Yaskawa INFORM job: SKRZYNIA_5140_0_STOPNI_2OBR_NEW.JBI

/JOB
//NAME SKRZYNIA_5140_0_STOPNI_2OBR_NEW
///FOLDERNAME 02-SKRZYNIE_JOBS
//POS
///NPOS 730,730,0,52,0,0
///TOOL 0
///POSTYPE PULSE
///PULSE
C00000=1055,-24125,84372,288,19725,204
C00001=0,-15438,65714,0,-68532,0
C00002=4718,-16587,59952,3396,-65485,-935
C00003=32997,-21499,42555,27623,-61436,21376
C00004=31759,-20688,42932,26837,-60850,21559
C00005=28987,-21156,42712,24818,-60442,22222
C00006=33447,-21964,42352,27886,-61721,21330
C00007=37687,-23357,41794,30651,-63289,20620
C00008=38979,-19018,48057,32961,-64962,20678
C00009=37261,-18075,48526,31902,-64209,20901
C00010=35830,-17198,48994,31015,-63571,21092
C00011=34080,-17614,48768,29780,-63290,21485
C00012=37261,-18075,48526,31902,-64209,20901
C00013=47373,-21912,40596,41149,-66086,26950
C00014=4718,-16587,59952,3396,-65485,-935
C00015=32997,-21499,42555,27623,-61436,21376
C00016=31759,-20688,42932,26837,-60850,21559
C00017=28987,-21156,42712,24818,-60442,22222
C00018=33447,-21964,42352,27886,-61721,21330
C00019=37687,-23357,41794,30651,-63289,20620
C00020=38979,-19018,48057,32961,-64962,20678
C00021=37261,-18075,48526,31902,-64209,20901
C00022=35830,-17198,48994,31015,-63571,21092
C00023=34080,-17614,48768,29780,-63290,21485
C00024=37261,-18075,48526,31902,-64209,20901
C00025=47373,-21912,40596,41149,-66086,26950
C00026=45033,-20851,41104,39798,-65001,27223
C00027=42790,-19693,41704,38494,-63946,27495
C00028=41070,-20182,41442,37324,-63566,27891
C00029=45033,-20851,41104,39798,-65001,27223
C00030=45033,-20851,41104,39798,-65001,27223
C00031=59624,-29540,14278,64846,-60867,16042
C00032=57357,-28542,14780,63940,-59509,16120
C00033=56188,-29140,14476,63237,-58995,16387
C00034=59588,-29370,14363,64862,-60819,16012
C00035=62924,-29779,15793,65870,-63073,16252
C00036=59724,-28781,16276,64511,-61238,16415
C00037=57764,-27936,16704,63709,-60078,16488
C00038=56408,-28589,16373,62897,-59486,16787
C00039=59724,-28781,16276,64511,-61238,16415
C00040=87562,-48087,-13810,78020,-75252,11220
C00041=10104,-46603,4759,11228,-37390,-5046
C00042=0,-52280,40443,0,6876,0
C00043=1529,-42140,58025,-5964,2417,3265
C00044=0,-38374,23626,-1605,-51738,268
C00045=45044,-23015,37260,35797,-71879,25522
C00046=39973,-29571,18873,35060,-63052,24165
C00047=38620,-28701,19269,34339,-62304,24363
C00048=36409,-29254,19014,32896,-61805,24958
C00049=44451,-29039,21934,37281,-65892,23702
C00050=49472,-39353,6917,53118,-50908,20251
C00051=45058,-39356,3832,51653,-47640,20099
C00052=42883,-38319,4163,50577,-46309,20295
C00053=40255,-38926,3967,48502,-45334,21060
C00054=46774,-39679,3737,52663,-48537,19827
C00055=48708,-40455,3517,53615,-49689,19657
C00056=43798,-39237,3871,50850,-47027,20335
C00057=41951,-38324,4161,49930,-45891,20507
C00058=39836,-38844,3994,48234,-45126,21137
C00059=48489,-40338,3551,53521,-49551,19665
C00060=48489,-40338,3551,53521,-49551,19665
C00061=44432,-39026,3936,51363,-47247,20139
C00062=42487,-38069,4248,50403,-46050,20315
C00063=39061,-38795,4009,47695,-44769,21310
C00064=44432,-39026,3936,51363,-47247,20139
C00065=45358,-49480,-3557,50155,-49322,21260
C00066=1817,-44984,2816,-3462,-45659,1296
C00067=1445,-28771,30219,-502,-63201,-220
C00068=1148,-56354,34370,-22,3827,-10
C00069=0,-52280,40443,0,6876,0
C00070=0,-49898,44897,0,-65513,0
C00071=52002,-27630,35066,40617,-70496,28619
C00072=38179,-24916,32897,32855,-63545,30206
C00073=36484,-23889,33369,31863,-62698,30449
C00074=33804,-24434,33113,30025,-62179,31112
C00075=38179,-24916,32897,32855,-63545,30206
C00076=78369,-41260,16071,67181,-65880,21417
C00077=137,-45861,52341,97,-67596,-14
C00078=-31499,-58302,-23356,15027,12889,-13082
C00079=-52768,-43016,-26078,18373,38595,-18774
C00080=-89470,-32103,-32973,29905,69139,-31512
C00081=-68838,-26884,-24872,16972,64732,-23076
C00082=-53036,-11528,-12218,12363,64665,-17409
C00083=-51536,-9474,-10276,11905,64649,-16876
C00084=-51739,-9114,-7787,12104,63269,-17104
C00085=-53036,-11528,-12218,12363,64665,-17409
C00086=-17541,-26226,-24397,927,59032,-5038
C00087=-17541,-26226,-24397,927,59032,-5038
C00088=-16950,-23991,-22741,715,59568,-4818
C00089=-17036,-23563,-20101,755,58071,-4857
C00090=-17541,-26226,-24397,927,59032,-5038
C00091=34102,-23192,-21614,-15638,64271,13209
C00092=33423,-21885,-20599,-15423,64418,12942
C00093=32426,-19856,-18975,-15106,64629,12551
C00094=32578,-19611,-17013,-15290,63535,12762
C00095=33423,-21885,-20599,-15423,64418,12942
C00096=59339,-6070,-6417,-20979,72191,20891
C00097=59339,-6070,-6417,-20979,72191,20891
C00098=57897,-4256,-4562,-20702,71913,20431
C00099=58108,-3992,-2506,-20878,70835,20713
C00100=59339,-6070,-6417,-20979,72191,20891
C00101=42744,-35904,-30225,-18322,62562,16651
C00102=-53036,-11528,-12218,12363,64665,-17409
C00103=-77982,-26538,-29134,27151,66629,-27745
C00104=-70983,-8594,-1966,26503,59809,-49670
C00105=-80152,19776,40785,37351,72704,-50428
C00106=-79984,20154,42529,37516,71911,-50638
C00107=-79233,18397,40079,37458,71885,-50340
C00108=-79984,20154,42529,37516,71911,-50638
C00109=-73519,23289,38838,28890,77081,-45618
C00110=-73519,24511,42682,29072,75582,-46027
C00111=-73519,23289,38838,28890,77081,-45618
C00112=-88897,15706,42282,50101,71325,-56974
C00113=-88897,15706,42282,50101,71325,-56974
C00114=-87612,12343,37838,50071,70996,-56519
C00115=-85283,14202,40272,50301,69633,-56165
C00116=-87338,12550,38107,50098,70839,-56476
C00117=-84952,-1789,13569,34660,47724,-58955
C00118=-67641,-1674,11109,10330,44856,-44725
C00119=-66443,961,13975,9688,44721,-44210
C00120=-67641,-1674,11109,10330,44856,-44725
C00121=-67641,-376,15347,10694,42950,-44967
C00122=-67641,-1674,11109,10330,44856,-44725
C00123=-79040,417,20398,15965,28992,-57786
C00124=-76655,5212,30978,15501,25024,-57306
C00125=-76655,6949,35816,16758,23084,-57955
C00126=-76655,5212,30978,15501,25024,-57306
C00127=-74761,6919,33010,13466,24593,-56049
C00128=-80460,-2874,12270,15804,32253,-57809
C00129=-61258,-29124,-13156,26560,43617,-22150
C00130=-30420,-40507,-29240,27153,53235,15188
C00131=-18589,-38725,-21450,23338,47896,18931
C00132=-17722,-35233,-16455,23322,46926,19051
C00133=-17722,-33749,-12435,23948,45421,18620
C00134=-17722,-33892,-12819,23887,45564,18661
C00135=-16677,-31133,-11209,23138,46167,19311
C00136=-17819,-35820,-17540,23246,47228,19090
C00137=-74104,-11494,-6266,31916,75042,4269
C00138=-71226,-7329,2631,32115,71468,4273
C00139=-71226,-6504,5446,32343,70365,3922
C00140=-71226,-6611,5086,32313,70505,3967
C00141=-68386,-4058,7675,32040,69573,4789
C00142=-73314,-9412,-353,32206,72648,3829
C00143=51751,-31069,-22965,-10739,49070,48663
C00144=49028,-23852,-11575,-9841,46366,47823
C00145=49028,-23004,-8935,-10039,45204,47956
C00146=49028,-23118,-9286,-10013,45357,47939
C00147=47000,-20813,-7527,-8928,45644,47024
C00148=50476,-26208,-15307,-10408,47325,48332
C00149=90602,-5375,6902,-38786,69848,59444
C00150=83174,19950,50269,-44999,67580,58220
C00151=82362,17902,47383,-44926,67511,57879
C00152=83515,19072,48341,-44798,68200,58056
C00153=78091,19382,40247,-36371,72286,52960
C00154=78091,20664,44011,-36670,70997,53443
C00155=78091,19382,40247,-36371,72286,52960
C00156=88699,7296,38566,-55615,63182,60372
C00157=86803,3068,32674,-55410,62638,59657
C00158=84852,4315,34115,-55564,61561,59330
C00159=86803,3068,32674,-55410,62638,59657
C00160=92770,-2803,21719,-53893,67577,59421
C00161=73393,-10627,10934,-27897,30744,62458
C00162=70789,-6606,18800,-27824,27830,62140
C00163=69654,-4593,20814,-26755,27596,61444
C00164=70789,-6606,18800,-27824,27830,62140
C00165=70789,-5070,23059,-29482,26284,63017
C00166=70789,-6606,18800,-27824,27830,62140
C00167=83486,-8736,6503,-27040,35338,66550
C00168=77831,-2041,26192,-25270,18452,68895
C00169=77967,1961,32070,-26860,17569,69698
C00170=77967,5243,40752,-32914,14549,72656
C00171=77967,1961,32070,-26860,17569,69698
C00172=74560,4730,35257,-21622,16551,66717
C00173=77967,1961,32070,-26860,17569,69698
C00174=81109,-22356,2664,-22493,33121,60116
C00175=86168,-49730,-13668,-23926,46819,49343
C00176=44183,-52048,-7537,-24795,46064,51426
C00177=0,-52280,40443,0,6876,0
C00178=0,-52280,40443,0,6876,0
C00179=33629,-57276,-6399,46271,-24969,-2804
C00180=75493,-63502,-64712,103874,-64610,-6298
C00181=47885,-58436,-62704,109755,-46164,-10686
C00182=43896,-60167,-65932,114356,-43302,-9311
C00183=55379,-67378,-68041,108237,-48773,-4935
C00184=62671,-64213,-64640,104431,-56093,-7372
C00185=28458,-50318,6850,47420,-25887,-3347
C00186=0,-52280,40443,0,6876,0
C00187=1055,-24125,84372,288,19725,204
C00188=0,-15438,65714,0,-68532,0
C00189=0,-15438,65714,966,-70097,42926
C00190=69988,-9219,57065,61610,-82752,27767
C00191=63113,-6157,59685,58080,-79692,28271
C00192=46673,-5697,67857,40481,-75278,29676
C00193=49770,-5379,67539,43594,-76189,29543
C00194=63113,-6157,59685,58080,-79692,28271
C00195=69988,-9219,57065,61610,-82752,27767
C00196=0,-15438,65714,966,-70097,42926
C00197=0,-15438,65714,0,-68532,0
C00198=1055,-24125,84372,288,19725,204
C00199=1055,-24125,84372,288,19725,204
C00200=0,-41971,13909,0,6774,1
C00201=-55064,-17017,13106,20113,45767,-35735
C00202=-85641,-3161,12660,31281,67420,-55579
C00203=-77611,9747,38455,32702,57795,-55547
C00204=-77611,9747,38455,32702,57795,-55547
C00205=-80481,23547,61641,37204,60115,-56891
C00206=-80479,11681,28780,33754,71138,-52780
C00207=-73572,15026,34389,33675,67405,-51294
C00208=-73572,20195,49236,35290,62248,-53161
C00209=-82806,26311,53816,38180,73291,-53604
C00210=-71695,3747,16001,30713,64750,-51022
C00211=-70421,5575,20105,30867,63066,-51036
C00212=-35543,-20105,-5144,22821,50284,-40173
C00213=-37830,-23193,-8618,23571,50957,-40982
C00214=11136,-28839,-12562,1025,41780,-20887
C00215=20486,-27077,-7346,-12554,38415,-10736
C00216=59545,-9921,5571,-27063,51925,3267
C00217=55110,-17412,-5825,-19778,50988,-2825
C00218=79390,11759,28162,-35512,71262,52960
C00219=74811,13878,33986,-35807,67493,52464
C00220=74942,18762,48004,-37392,62815,54352
C00221=76815,18630,46530,-37158,64288,54543
C00222=79390,11759,28162,-35512,71262,52960
C00223=10831,-54278,-29128,-6468,39852,-5090
C00224=-67200,-10549,24402,-3189,24913,-39001
C00225=-75122,-2194,12822,3152,39225,-43427
C00226=-77516,10189,32861,8493,33365,-45533
C00227=-75154,17575,49272,7885,27457,-44928
C00228=-68113,9932,38901,1157,28472,-40453
C00229=-67114,5383,31515,9208,32648,-43213
C00230=-66450,3998,29285,10896,33890,-43630
C00231=-66374,3101,28136,14657,35566,-44954
C00232=-66576,452,24763,27028,43375,-49112
C00233=-69928,4230,30673,35488,50431,-52676
C00234=-77050,-3138,8526,33226,61087,-51698
C00235=-67200,-10549,24402,-3189,24913,-39001
C00236=0,-52280,40443,83103,28146,-16510
C00237=99993,-20782,22705,-13349,24734,56519
C00238=67200,-10549,24402,3189,24913,39001
C00239=75122,-2194,12822,-3152,39225,43427
C00240=74323,5203,27259,-5972,33194,43789
C00241=74015,16414,48063,-6821,27325,44224
C00242=56519,1138,28747,9235,29393,33453
C00243=55467,619,28251,10155,29461,32830
C00244=56374,-724,25854,4078,30541,35419
C00245=56480,-7201,15910,-17697,38451,43334
C00246=68252,956,25699,-34035,49810,51639
C00247=77050,-3138,8526,-33226,61087,51698
C00248=67200,-10549,24402,3189,24913,39001
C00249=0,-52280,40443,-83103,28146,16510
C00250=-99993,-20782,22705,13349,24734,-56519
C00251=-91125,453,39555,30378,52425,-51131
C00252=-81425,-5449,14825,37552,56592,-47667
C00253=-81425,-10835,-2515,34915,62871,-45127
C00254=-79239,4305,16082,37593,68846,-50182
C00255=-81302,5892,27588,46359,62943,-54679
C00256=-82227,19402,59913,51524,57300,-60581
C00257=-84844,8890,27031,38640,69740,-53449
C00258=-90096,4679,14083,37467,76581,-51973
C00259=-87885,29238,52923,40761,81198,69685
C00260=-84355,23847,39024,40698,83720,72224
C00261=-81960,27335,46957,41070,80536,71891
C00262=-82643,24718,50492,48951,72637,70260
C00263=-90480,18737,31939,47254,81986,71631
C00264=-94217,10634,17426,46901,86469,-59967
C00265=-81425,-10835,-2515,34915,62871,-45127
C00266=-81425,-5449,14825,37552,56592,-47667
C00267=-94290,-610,44819,32366,49686,-53459
C00268=0,-55136,17047,60468,32096,-4233
C00269=99993,-20782,22705,-13349,24734,56519
C00270=91125,453,39555,-30378,52425,51131
C00271=81425,-5449,14825,-37552,56592,47667
C00272=81425,-10835,-2515,-34915,62871,45127
C00273=79239,4305,16082,-37593,68846,50182
C00274=83239,4964,30263,-50637,62037,57149
C00275=83991,16425,61235,-57769,55250,63273
C00276=93928,7973,40920,-53095,64494,61640
C00277=75109,22299,39152,-26915,78743,47998
C00278=79256,17348,34699,-33448,76412,88212
C00279=79932,23608,50901,-39863,71219,88955
C00280=76220,30771,63034,-41386,67395,88927
C00281=86322,16060,37848,-39554,76452,89287
C00282=87424,-1569,9538,-38190,72401,52253
C00283=81425,-10835,-2515,-34915,62871,45127
C00284=92850,-11266,9233,-39092,60986,50964
C00285=28366,-40369,19479,-5635,23506,17663
C00286=-80334,-19501,31260,21216,42469,-40219
C00287=-80621,-32280,-9061,25825,59412,-41877
C00288=-80621,-37319,-22868,24573,64555,-40576
C00289=-75108,-2453,16462,35304,60348,-42510
C00290=-72231,7240,33473,36511,55681,-43130
C00291=-35770,-19109,7486,28512,40799,-31761
C00292=-39606,-22901,-1163,28356,44724,-32188
C00293=15344,-29112,-5358,-2858,33820,-6852
C00294=13390,-24012,2637,-1527,32105,-7853
C00295=57983,-8601,15571,-27088,42703,12849
C00296=60973,-17187,4937,-27817,44388,13718
C00297=60973,-17187,4937,-27817,44388,13718
C00298=-13287,-42463,-12044,19170,31021,-23010
C00299=-17374,-21287,20534,22794,29118,-26096
C00300=13276,-20759,18622,-1911,29377,-7028
C00301=39924,-14247,19329,-14795,35999,4396
C00302=41528,-14133,18797,-15449,36702,5040
C00303=57001,-5890,26499,-21893,40771,11494
C00304=64054,-19541,3059,-29141,44956,15011
C00305=51466,-33957,-1499,-46586,51805,23434
C00306=17032,-20770,22044,-28854,30468,11088
C00307=-9868,-18638,14971,-8492,38486,-5199
C00308=-40562,-13194,19800,9508,35447,-20184
C00309=-41848,-12620,20103,10165,35810,-20773
C00310=-57278,-4046,28217,17578,39066,-27653
C00311=-71680,-19835,10874,33863,39440,-36917
C00312=-20806,-37586,-12792,9951,42782,-18031
C00313=29087,-45372,27330,-13325,19529,9021
C00314=0,-52280,40443,0,6876,0
C00315=0,-52280,40443,0,6876,0
C00316=0,-17525,61946,0,273,32004
C00317=54446,-4421,37881,-48560,57645,57448
C00318=45059,-5790,38757,-53071,45868,54447
C00319=46561,-4822,57063,-86189,40693,71736
C00320=46137,-328,57206,-69896,42561,59838
C00321=35508,-2998,35633,-40347,47515,38753
C00322=43067,2853,36106,-38598,60324,43004
C00323=45059,-5790,38757,-53071,45868,54447
C00324=54446,-4421,37881,-48560,57645,57448
C00325=0,-17525,61946,0,273,32004
C00326=0,-52280,40443,0,6876,0
C00327=0,-52280,40443,0,6876,0
C00328=0,-52280,40443,0,6876,0
C00329=0,-52280,40443,0,-42737,40640
C00330=0,-52280,40443,0,-42737,40640
C00331=64551,-35409,28076,75550,-44539,17239
C00332=49799,-25338,45366,61341,-39751,21495
C00333=45731,-22710,35392,68644,-36821,18294
C00334=37993,-24684,30723,57032,-36974,21705
C00335=37887,-25651,28733,57662,-36597,21303
C00336=43117,-27612,29118,67655,-35359,18183
C00337=39863,-22026,47404,54615,-35502,22403
C00338=0,-52277,40442,0,6872,2
C00339=0,-38538,66749,0,-898,0
C00340=0,-52280,40443,0,-79033,35417
C00341=46775,-35113,22190,42926,-67531,20697
C00342=52587,-26056,25345,47610,-66542,17970
C00343=45640,-25642,24411,43945,-63126,18913
C00344=46067,-27754,19531,44807,-62059,18176
C00345=53914,-29436,22058,48262,-67266,17843
C00346=63113,-6157,59685,58080,-79692,28271
C00347=47789,-6280,67353,41142,-75661,29541
C00348=46856,-5642,67903,40595,-75324,29647
C00349=49398,-5231,67705,43314,-76061,29572
C00350=59203,-5425,63284,53118,-78384,28542
C00351=46775,-35113,22190,42926,-67531,20697
C00352=0,-52280,40443,0,-79033,35417
C00353=0,-52280,40443,0,-61239,28081
C00354=53819,-14110,13758,-46164,60155,50576
C00355=48398,-14119,9451,-44868,59619,48162
C00356=41231,-18689,20734,-60860,39616,53092
C00357=26205,-20881,5343,-31434,40895,31963
C00358=48398,-14119,9451,-44868,59619,48162
C00359=53819,-14110,13758,-46164,60155,50576
C00360=0,-52280,40443,0,-61239,28081
C00361=404,-42897,57020,-1574,2523,869
C00362=404,-42897,57020,-1574,2523,869
C00363=0,-52280,40443,0,6876,0
C00364=-99253,-13690,44082,59847,13407,-31313
C00365=-87814,-12734,20141,45739,-14352,-64418
C00366=-86669,-6582,30812,41148,-16781,-62025
C00367=-85055,-5827,31548,44003,-17420,-63187
C00368=-85971,-6262,31124,42409,-17052,-62539
C00369=-86650,-5303,32069,41395,-16716,-62141
C00370=-94954,-14494,-1860,-7818,15857,-59130
C00371=-93142,-9291,12181,-6959,15791,-58178
C00372=-93142,-8228,15250,-7572,14488,-57881
C00373=-93142,-9291,12181,-6959,15791,-58178
C00374=-86125,-12470,22545,29004,-25567,-58412
C00375=-83883,-11340,22525,32952,-25567,-60136
C00376=-82768,-10824,22986,34487,-25904,-60776
C00377=-83883,-11340,22525,32952,-25567,-60136
C00378=-85143,-9772,23941,31487,-24966,-59556
C00379=-83883,-11340,22525,32952,-25567,-60136
C00380=-85732,-21202,11427,30682,-24763,-59235
C00381=-84150,-10929,23786,31981,-25941,-59678
C00382=-83036,-10419,24246,33504,-26268,-60308
C00383=-84150,-10929,23786,31981,-25941,-59678
C00384=-85291,-9507,25078,30650,-25411,-59154
C00385=-84150,-10929,23786,31981,-25941,-59678
C00386=-85786,-16909,14677,31743,-23900,-59790
C00387=-84150,-10498,24888,31517,-26306,-59436
C00388=-83174,-10052,25293,32841,-26587,-59984
C00389=-84150,-10498,24888,31517,-26306,-59436
C00390=-85258,-9112,26156,30226,-25800,-58928
C00391=-84150,-10498,24888,31517,-26306,-59436
C00392=-87841,-18519,13420,28367,-23534,-58339
C00393=-84845,-10773,24694,30524,-26144,-59020
C00394=-83241,-10052,25348,32714,-26598,-59924
C00395=-84150,-10465,24972,31484,-26336,-59417
C00396=-85145,-9228,26102,30329,-25881,-58963
C00397=-84150,-10465,24972,31484,-26336,-59417
C00398=-86371,-18277,13606,30568,-23951,-59265
C00399=-84931,-11946,21758,31628,-25145,-59609
C00400=-83211,-11173,22442,34044,-25650,-60618
C00401=-84345,-11688,21985,32461,-25312,-59957
C00402=-85283,-10526,23025,31366,-24861,-59525
C00403=-84345,-11688,21985,32461,-25312,-59957
C00404=-86191,-19647,12567,30467,-24278,-59187
C00405=-84870,-11108,23866,30820,-25860,-59178
C00406=-83051,-10286,24607,33321,-26381,-60213
C00407=-84345,-10877,24073,31552,-26006,-59481
C00408=-85179,-9842,25009,30582,-25619,-59100
C00409=-84345,-10877,24073,31552,-26006,-59481
C00410=-85438,-18022,14839,31140,-24818,-59429
C00411=-84247,-11820,22550,32049,-25753,-59727
C00412=-84627,-11209,23435,31382,-25751,-59435
C00413=-82990,-10465,24105,33639,-26227,-60372
C00414=-84104,-10976,23642,32111,-25899,-59738
C00415=-84898,-9998,24525,31196,-25529,-59378
C00416=-84104,-10976,23642,32111,-25899,-59738
C00417=-86610,-16845,14732,30573,-23614,-59301
C00418=-84466,-11025,23783,31488,-25891,-59466
C00419=-82824,-10273,24459,33737,-26370,-60397
C00420=-84104,-10864,23927,31990,-25993,-59674
C00421=-84789,-10021,24690,31200,-25673,-59363
C00422=-84104,-10864,23927,31990,-25993,-59674
C00423=-83806,-19585,12613,33764,-25080,-60559
C00424=-84285,-10368,25328,31127,-26432,-59250
C00425=-82780,-9675,25960,33156,-26866,-60087
C00426=-83924,-10205,25475,31619,-26533,-59453
C00427=-84478,-9530,26093,30986,-26280,-59206
C00428=-83924,-10205,25475,31619,-26533,-59453
C00429=-87149,-17993,13826,29513,-23647,-58830
C00430=-84920,-13182,20975,31162,-25481,-59361
C00431=-84012,-10708,24730,31646,-26390,-59479
C00432=-82779,-10142,25241,33309,-26748,-60166
C00433=-83711,-10572,24852,32056,-26475,-59649
C00434=-84370,-9774,25579,31305,-26170,-59356
C00435=-83711,-10572,24852,32056,-26475,-59649
C00436=-83642,-3679,42021,23358,-36761,-56118
C00437=-85886,-5975,41264,18964,-40261,-54782
C00438=-84505,-11891,22094,31989,-25448,-59736
C00439=-82884,-11162,22742,34234,-25925,-60671
C00440=-83919,-11632,22322,32811,-25616,-60079
C00441=-84723,-10654,23196,31887,-25230,-59715
C00442=-83919,-11632,22322,32811,-25616,-60079
C00443=-87348,-16035,7353,17528,-35245,-56477
C00444=-86906,-16205,7213,17977,-35365,-56684
C00445=-86616,-16813,3502,19256,-33445,-57386
C00446=-85308,-16228,3988,20718,-33648,-58082
C00447=-86244,-16649,3638,19674,-33501,-57585
C00448=-86740,-15973,4201,19194,-33277,-57362
C00449=-86244,-16649,3638,19674,-33501,-57585
C00450=-73780,-8639,20128,34258,-51705,-52097
C00451=-90965,-18271,-29411,11001,-28333,-56925
C00452=-93309,-19947,-33502,6140,-24593,-56497
C00453=-91512,-19116,-32812,8551,-24603,-57834
C00454=-92565,-19610,-33223,7138,-24591,-57051
C00455=-93003,-18716,-32476,6600,-24397,-56752
C00456=-92565,-19610,-33223,7138,-24591,-57051
C00457=-92565,-19610,-33223,7138,-24591,-57051
C00458=-95836,-54375,-51122,6031,-17685,-48210
C00459=-95836,-54375,-51122,6031,-17685,-48210
C00460=-43821,-47238,-2775,-3022,56549,-3681
C00461=-20126,-26882,59542,2406,16879,-9162
C00462=-20126,-26882,59542,2406,16879,-9162
C00463=98601,-10520,92678,4674,-40855,-9615
C00464=95537,-19831,-2695,-2933,-44471,35837
C00465=92548,-20391,-28429,-6186,-30623,55200
C00466=93192,-17848,-29686,-6005,-27810,55077
C00467=92147,-17363,-29270,-7221,-27815,55772
C00468=90371,-16495,-28521,-9286,-27856,56953
C00469=91429,-17018,-28974,-8057,-27827,56250
C00470=92033,-15799,-27911,-7415,-27588,55880
C00471=91429,-17018,-28974,-8057,-27827,56250
C00472=92548,-20391,-28429,-6186,-30623,55200
C00473=91156,-15018,-4648,-8036,-38181,54813
C00474=90585,-14766,-4428,-8565,-38201,55100
C00475=88830,-13959,-3717,-10186,-38284,55977
C00476=89897,-14456,-4157,-9202,-38230,55445
C00477=90761,-12944,-2809,-8452,-37927,55043
C00478=89897,-14456,-4157,-9202,-38230,55445
C00479=89910,-11217,67535,-9455,-58896,55399
C00480=89910,-11217,67535,-9455,-58896,55399
C00481=85786,-16735,14816,-31782,-23869,59812
C00482=84033,-13230,17727,-35008,-23968,61233
C00483=82251,-12406,18443,-37550,-24551,62308
C00484=83514,-12996,17929,-35760,-24132,61552
C00485=84258,-12095,18717,-34917,-23742,61217
C00486=83514,-12996,17929,-35760,-24132,61552
C00487=87149,-17993,13826,-29513,-23647,58830
C00488=83574,-13027,17908,-35676,-24115,61514
C00489=81915,-12248,18589,-38020,-24666,62504
C00490=83118,-12818,18089,-36330,-24263,61791
C00491=83897,-11882,18912,-35460,-23856,61445
C00492=83118,-12818,18089,-36330,-24263,61791
C00493=83806,-19585,12613,-33764,-25080,60559
C00494=83575,-13270,17698,-35618,-24145,61476
C00495=81675,-12378,18472,-38297,-24777,62607
C00496=82998,-13006,17925,-36445,-24332,61826
C00497=83876,-11958,18841,-35466,-23874,61442
C00498=82998,-13006,17925,-36445,-24332,61826
C00499=86610,-16845,14732,-30573,-23614,59301
C00500=82990,-13468,17528,-36367,-24395,61793
C00501=81406,-12724,18174,-38578,-24928,62723
C00502=82493,-13239,17725,-37070,-24559,62089
C00503=83436,-12134,18690,-36041,-24064,61684
C00504=82493,-13239,17725,-37070,-24559,62089
C00505=84814,-16043,15376,-33312,-24093,60464
C00506=83076,-13850,17202,-36172,-24411,61704
C00507=81384,-13062,17878,-38534,-24974,62698
C00508=82555,-13613,17404,-36910,-24580,62015
C00509=83566,-12434,18427,-35805,-24047,61580
C00510=82555,-13613,17404,-36910,-24580,62015
C00511=86191,-19647,12567,-30467,-24278,59187
C00512=83141,-13940,17126,-36065,-24398,61655
C00513=81467,-13161,17792,-38413,-24955,62645
C00514=82500,-13648,17375,-36975,-24607,62039
C00515=83481,-12505,18364,-35905,-24087,61617
C00516=82500,-13648,17375,-36975,-24607,62039
C00517=86371,-18277,13606,-30568,-23951,59265
C00518=83407,-14016,17058,-35697,-24309,61505
C00519=81715,-13237,17726,-38081,-24865,62509
C00520=82904,-13790,17251,-36416,-24470,61808
C00521=83686,-12878,18037,-35556,-24055,61469
C00522=82904,-13790,17251,-36416,-24470,61808
C00523=87841,-18519,13420,-28367,-23534,58339
C00524=83373,-14160,16936,-35712,-24341,61507
C00525=81692,-13388,17594,-38077,-24893,62505
C00526=82748,-13879,17174,-36603,-24542,61883
C00527=83607,-12881,18032,-35663,-24082,61515
C00528=82748,-13879,17174,-36603,-24542,61883
C00529=85786,-16909,14677,-31743,-23900,59790
C00530=83147,-14479,16665,-35944,-24472,61597
C00531=81460,-13708,17319,-38301,-25026,62591
C00532=82520,-14198,16902,-36833,-24674,61972
C00533=83571,-12989,17938,-35691,-24113,61524
C00534=82520,-14198,16902,-36833,-24674,61972
C00535=85732,-21202,11427,-30682,-24763,59235
C00536=83169,-14709,16474,-35859,-24497,61553
C00537=81172,-13798,17245,-38643,-25153,62725
C00538=82398,-14365,16763,-36952,-24745,62014
C00539=83600,-12984,17944,-35650,-24102,61504
C00540=82398,-14365,16763,-36952,-24745,62014
C00541=92346,-18713,13565,-21110,-22545,55257
C00542=83258,-14188,16907,-35850,-24389,61565
C00543=81518,-13384,17592,-38292,-24965,62594
C00544=82794,-13980,17083,-36511,-24538,61844
C00545=83714,-12912,18003,-35501,-24048,61445
C00546=82794,-13980,17083,-36511,-24538,61844
C00547=86140,-12802,12665,-93523,-10743,85795
C00548=86837,-13114,12391,-93393,-10290,85805
C00549=85030,-12289,13120,-93723,-11463,85776
C00550=86140,-12802,12665,-93523,-10743,85795
C00551=86958,-11660,13681,-94506,-10238,86349
C00552=85239,-16743,-4327,42764,21357,45785
C00553=86298,-7639,7084,25531,26453,52172
C00554=86298,-6383,11028,27162,24874,51322
C00555=86298,-7639,7084,25531,26453,52172
C00556=82295,-26986,-30576,21875,37939,54070
C00557=85045,-36869,-4353,-28502,-22832,52282
C00558=0,-24029,84339,0,19981,0
C00559=0,-24029,84339,0,19981,0
C00560=3172,-24246,80980,3465,15913,689
C00561=-86563,-26985,13879,10257,-21548,-45530
C00562=-86191,-19647,12567,30467,-24278,-59187
C00563=-83221,-13587,17636,37793,-25116,-62228
C00564=-91978,-13833,14560,12391,-18633,-51524
C00565=-94992,-13830,14285,1276,-18012,-46664
C00566=-84074,-17488,11256,38660,-23649,-62784
C00567=-73679,-33270,1000,44272,-31600,-64253
C00568=-86926,-60758,23267,6576,1160,-9545
C00569=0,-52280,40443,0,6876,0
C00570=82475,-58079,26734,835,4084,4444
C00571=97932,-26840,7691,8784,-23444,42538
C00572=87166,-16607,16322,-25365,-24201,56345
C00573=84744,-11374,21734,-29079,-24723,57922
C00574=84804,-11023,22730,-28561,-25071,57659
C00575=85100,-26994,10417,-24982,-28140,55821
C00576=0,-52280,40443,0,6876,0
C00577=0,-52280,40443,0,6876,0
C00578=-90140,-60305,18108,-2708,1721,-7625
C00579=-95594,-27428,6866,-4663,-19832,-42154
C00580=-98688,-13767,16447,-18366,-10080,-35766
C00581=-99366,-12207,13361,-76262,-4504,-7609
C00582=-98825,-14297,3352,-138105,-6872,21732
C00583=-99703,-3544,30885,-62667,-5630,-13378
C00584=-99859,-2424,20650,-157436,-17585,31647
C00585=-99057,-6525,-3028,-166156,-45024,38419
C00586=-98286,-5427,328,-166417,-43477,38616
C00587=-98488,3848,8620,-169322,-45735,38851
C00588=-99936,2884,1652,-167416,-53424,38690
C00589=-96149,-9016,-15084,-169449,-55688,40292
C00590=-90140,-60305,18108,-2708,1721,-7625
C00591=0,-52280,40443,0,6876,0
C00592=84259,-57935,27522,-3761,3673,6310
C00593=86507,-39672,4297,-27618,-16640,46340
C00594=73669,-37119,-20783,-92053,-19719,85232
C00595=86539,-20830,1725,-71850,-11773,76853
C00596=97574,-21911,-7032,-15733,6173,47170
C00597=94640,-18033,-2805,930,6039,39142
C00598=97727,-14050,2363,-13742,12741,47040
C00599=100679,-6296,-4637,-9974,40184,43946
C00600=100653,-5025,-17306,-8356,57963,47370
C00601=98357,-1060,-14638,-7161,64336,49394
C00602=99096,-3774,-7192,-7126,47828,42427
C00603=97072,-20012,-39240,-5169,57466,41015
C00604=96250,-19428,-8283,-4838,27297,37910
C00605=86507,-39672,4297,-27618,-16640,46340
C00606=84259,-57935,27522,-3761,3673,6310
C00607=0,-52280,40443,0,6876,0
C00608=0,-27933,77061,0,20812,0
C00609=0,-27933,77061,0,20812,0
C00610=0,-52280,40443,0,6876,0
C00611=-91970,-60791,14435,-3343,512,-9412
C00612=-98647,-24138,10005,-11519,-21203,-39749
C00613=-99883,-13980,22886,-11640,-25090,-40341
C00614=-99702,-9154,61728,-1148,-61809,-40243
C00615=-84328,-13042,29707,23458,-33731,-54641
C00616=-83101,-4179,39208,25894,-34785,-55667
C00617=-82881,-4330,38692,26392,-34479,-55866
C00618=-76259,-18287,26646,31659,-38322,-57579
C00619=-89741,-28009,12101,4461,-28076,-46404
C00620=-91970,-60791,14435,-3343,512,-9412
C00621=0,-52280,40443,0,6876,0
C00622=91083,-60784,14823,-9043,-825,15173
C00623=83869,-19403,12921,-33769,-24740,60260
C00624=83869,-19403,12921,-33769,-24740,60260
C00625=83932,-19538,53415,-33663,-71112,60249
C00626=83932,-19538,53415,-33663,-71112,60249
C00627=82480,-12247,21118,-35440,-26416,60009
C00628=82194,-11433,19802,-37650,-25323,61125
C00629=81904,-9374,24711,-35791,-26879,60109
C00630=79790,-20261,14917,-36681,-28829,60258
C00631=76554,-29711,-1870,-46042,-25952,65654
C00632=91083,-60784,14823,-9043,-825,15173
C00633=0,-52280,40443,0,6876,0
C00634=-91526,-60598,16699,7584,176,-13289
C00635=-81382,-25890,9219,35455,-25500,-59095
C00636=-86453,-20958,12525,30076,-22568,-57089
C00637=-86589,-16097,16237,31250,-21582,-57704
C00638=-98933,-11298,20505,-13970,-18736,-37953
C00639=-98281,-10965,21163,-11559,-18548,-39330
C00640=-85424,-18472,14402,34409,-22969,-58895
C00641=-74746,-27148,8488,44263,-29128,-62418
C00642=-81326,-27507,8265,35533,-26282,-59001
C00643=-91415,-60262,16631,7870,-73,-13734
C00644=24,-24029,84339,7,19981,5
C00645=100404,-52373,45687,-1822,14816,-5144
C00646=75939,-26469,7919,-40869,-29645,63133
C00647=81882,-22565,10470,-35355,-26404,61107
C00648=82801,-12246,21732,-34208,-26055,60642
C00649=91782,-10629,23559,-8729,-22207,49851
C00650=96500,-9524,26299,5706,-23134,43728
C00651=77262,-23244,14300,-38922,-31295,61912
C00652=78410,-22868,15324,-38001,-30064,61274
C00653=96357,-43275,13317,73005,-20942,3046
C00654=567,-24029,84339,168,19981,112
C00655=-91970,-60791,14435,-3343,512,-9412
C00656=-98991,-22833,11519,-12824,-17638,-36336
C00657=-86376,-13627,18436,38326,-18406,-58533
C00658=-85581,-10814,20279,41280,-18093,-59893
C00659=-85472,-10371,21054,41064,-18287,-59771
C00660=-86274,-24518,9978,34497,-20333,-56613
C00661=-91684,-53777,2301,20525,-9313,-33684
C00662=-67305,-55044,34987,1504,5690,-2468
C00663=0,-52280,40443,0,6876,0
C00664=77036,-56616,31288,-2531,4707,4197
C00665=84359,-28321,8817,-32860,-20485,54199
C00666=81156,-16932,14874,-39538,-26422,62851
C00667=93153,-15089,13046,-5673,-18101,48746
C00668=90780,-14174,15526,-13510,-19626,52025
C00669=77970,-27630,4721,-41834,-28549,63607
C00670=81111,-35571,7141,-33980,-21909,52006
C00671=82626,-57814,28323,-4146,3364,6346
C00672=0,-52280,40443,0,6876,0
C00673=0,-28135,76691,0,20839,0
C00674=0,-28135,76691,0,20839,0
C00675=-45332,-39712,59352,-1730,18713,2903
C00676=-94065,-8316,59352,-1730,-37754,-40387
C00677=-100331,-14895,33931,-8215,-36518,-40227
C00678=-98931,-8578,39429,-6260,-48307,-43744
C00679=-100336,-4176,46216,-7600,-55875,-44633
C00680=-93952,8947,73671,995,-68520,-43850
C00681=-98791,-3170,32594,-4861,-60761,-43748
C00682=-98640,4466,38023,-4864,-58745,-43707
C00683=-98715,-12714,-17812,-7609,-33367,-41875
C00684=-98688,-14490,-28435,-9054,-27450,-41090
C00685=-99605,-15546,-21493,-8548,-33053,-41326
C00686=-100467,-8208,-2562,-8095,-44661,-42156
C00687=-93952,8947,73671,995,-68520,-43850
C00688=-88754,54,62805,4404,-67858,-45120
C00689=-100222,-4532,45667,-7492,-55263,-44561
C00690=-100331,-14895,33931,-8215,-36518,-40227
C00691=-94065,-8316,59352,-1730,-37754,-40387
C00692=-45544,-32973,71870,-2133,15168,3033
C00693=0,-28135,76691,0,20839,0
C00694=54178,-17846,77779,596,-29686,20997
C00695=54178,-17846,77779,596,-29686,20997
C00696=99462,-18987,75418,611,-28919,20989
C00697=98707,-9390,78674,1080,-71212,38250
C00698=98768,-5182,41096,1808,-44974,38308
C00699=100431,1771,51615,3823,-56746,39115
C00700=97953,-6621,17555,2289,-50176,39420
C00701=95834,-5353,18817,760,-50052,40242
C00702=86491,-3931,18489,-13403,-48438,44853
C00703=88887,-11110,-8515,-11527,-36861,46615
C00704=88808,-13839,-20865,-13699,-30585,47852
C00705=90457,-16080,-12990,-9972,-37305,45724
C00706=97953,-6621,17555,2289,-50176,39420
C00707=100431,1771,51615,3823,-56746,39115
C00708=98768,-5182,41096,1808,-44974,38308
C00709=98707,-9390,78674,1080,-71212,38250
C00710=0,-28135,76691,0,20839,0
C00711=0,-28135,76691,0,20839,0
C00712=-91526,-60598,16699,7584,176,-13289
C00713=-81382,-25890,9219,35455,-25500,-59095
C00714=-81382,-25890,9219,35455,-25500,-59095
C00715=-85509,-13950,19358,32213,-22393,-58041
C00716=-96341,-12086,19487,-5053,-17846,-42145
C00717=-97523,-9822,24708,-8570,-19966,-40659
C00718=-84656,-25369,12054,31249,-26195,-57129
C00719=-82652,-57346,29982,2770,3944,-5064
C00720=0,-52280,40443,0,6876,0
C00721=60653,-54633,35892,-1212,5841,2035
C00722=77942,-28227,6869,-38010,-29303,61907
C00723=82500,-13648,17375,-36975,-24607,62039
C00724=80844,-11529,18736,-41531,-25394,63903
C00725=80409,-10373,22284,-40214,-26848,63104
C00726=64389,-31987,5108,-50419,-37074,66126
C00727=60653,-54633,35892,-1212,5841,2035
C00728=0,-52280,40443,0,6876,0
C00729=0,-28167,76633,0,20843,0
BC00000=413138
BC00001=413138
BC00002=295997
BC00003=264574
BC00004=264574
BC00005=264574
BC00006=264574
BC00007=233852
BC00008=284288
BC00009=284288
BC00010=284288
BC00011=284288
BC00012=284288
BC00013=356545
BC00014=388163
BC00015=356740
BC00016=356740
BC00017=356740
BC00018=356740
BC00019=356740
BC00020=407176
BC00021=407176
BC00022=407176
BC00023=407176
BC00024=407176
BC00025=479433
BC00026=479433
BC00027=479433
BC00028=479433
BC00029=479433
BC00030=530237
BC00031=530237
BC00032=530237
BC00033=530237
BC00034=530237
BC00035=601977
BC00036=601977
BC00037=601977
BC00038=601977
BC00039=601977
BC00040=601977
BC00041=522422
BC00042=522422
BC00043=671734
BC00044=689202
BC00045=689202
BC00046=689202
BC00047=689202
BC00048=689202
BC00049=689202
BC00050=726463
BC00051=726463
BC00052=726463
BC00053=726463
BC00054=726463
BC00055=782137
BC00056=782137
BC00057=782137
BC00058=782137
BC00059=782137
BC00060=850421
BC00061=850421
BC00062=850421
BC00063=850421
BC00064=850421
BC00065=850421
BC00066=823841
BC00067=797607
BC00068=755227
BC00069=755227
BC00070=915219
BC00071=914226
BC00072=914226
BC00073=914226
BC00074=914226
BC00075=914226
BC00076=914226
BC00077=922367
BC00078=927819
BC00079=927819
BC00080=927819
BC00081=943180
BC00082=943180
BC00083=943180
BC00084=943180
BC00085=943180
BC00086=943180
BC00087=943180
BC00088=943180
BC00089=943180
BC00090=943180
BC00091=943180
BC00092=943180
BC00093=943180
BC00094=943180
BC00095=943180
BC00096=943180
BC00097=943180
BC00098=943180
BC00099=943180
BC00100=943180
BC00101=943180
BC00102=943180
BC00103=943180
BC00104=943180
BC00105=943180
BC00106=943182
BC00107=943182
BC00108=943182
BC00109=943182
BC00110=943182
BC00111=943182
BC00112=943182
BC00113=943182
BC00114=943182
BC00115=943182
BC00116=943182
BC00117=943182
BC00118=943182
BC00119=943182
BC00120=943182
BC00121=943182
BC00122=943182
BC00123=943182
BC00124=943182
BC00125=943182
BC00126=943182
BC00127=943182
BC00128=943182
BC00129=943183
BC00130=943184
BC00131=943184
BC00132=943184
BC00133=943184
BC00134=943184
BC00135=943184
BC00136=943184
BC00137=943184
BC00138=943184
BC00139=943184
BC00140=943184
BC00141=943156
BC00142=943170
BC00143=943170
BC00144=943170
BC00145=943170
BC00146=943170
BC00147=943170
BC00148=943170
BC00149=943184
BC00150=943184
BC00151=943184
BC00152=943184
BC00153=943184
BC00154=943184
BC00155=943184
BC00156=943184
BC00157=943184
BC00158=943184
BC00159=943184
BC00160=943184
BC00161=943184
BC00162=943184
BC00163=943184
BC00164=943184
BC00165=943184
BC00166=943184
BC00167=943184
BC00168=943184
BC00169=943184
BC00170=943184
BC00171=943184
BC00172=943184
BC00173=943184
BC00174=911399
BC00175=884954
BC00176=838173
BC00177=838173
BC00178=727925
BC00179=734552
BC00180=750834
BC00181=750837
BC00182=811927
BC00183=811927
BC00184=760768
BC00185=744267
BC00186=744267
BC00187=413138
BC00188=413138
BC00189=413138
BC00190=408626
BC00191=408626
BC00192=408753
BC00193=347392
BC00194=408626
BC00195=408626
BC00196=413138
BC00197=413138
BC00198=413138
BC00199=505502
BC00200=893917
BC00201=915147
BC00202=918406
BC00203=918406
BC00204=918406
BC00205=918406
BC00206=935268
BC00207=935270
BC00208=935270
BC00209=935270
BC00210=935270
BC00211=935270
BC00212=935270
BC00213=935270
BC00214=935270
BC00215=935269
BC00216=935270
BC00217=935271
BC00218=935271
BC00219=935271
BC00220=935271
BC00221=935271
BC00222=935271
BC00223=930781
BC00224=906929
BC00225=936106
BC00226=936109
BC00227=936109
BC00228=936106
BC00229=936107
BC00230=936108
BC00231=936108
BC00232=936109
BC00233=936109
BC00234=936109
BC00235=906929
BC00236=835535
BC00237=835535
BC00238=906929
BC00239=936106
BC00240=936109
BC00241=936109
BC00242=936109
BC00243=936109
BC00244=936114
BC00245=936121
BC00246=936110
BC00247=936109
BC00248=906929
BC00249=835535
BC00250=835535
BC00251=872997
BC00252=918800
BC00253=938197
BC00254=938199
BC00255=938199
BC00256=938199
BC00257=938199
BC00258=938775
BC00259=938199
BC00260=952138
BC00261=952138
BC00262=952138
BC00263=952138
BC00264=952138
BC00265=938197
BC00266=918800
BC00267=872997
BC00268=873283
BC00269=835535
BC00270=872997
BC00271=918800
BC00272=938197
BC00273=938199
BC00274=938199
BC00275=938199
BC00276=938199
BC00277=938199
BC00278=938199
BC00279=938199
BC00280=938199
BC00281=938199
BC00282=938199
BC00283=938197
BC00284=918800
BC00285=849812
BC00286=864290
BC00287=883850
BC00288=922155
BC00289=922155
BC00290=922155
BC00291=922153
BC00292=922155
BC00293=922155
BC00294=922155
BC00295=922153
BC00296=922155
BC00297=914820
BC00298=922155
BC00299=922155
BC00300=922151
BC00301=922153
BC00302=922197
BC00303=922153
BC00304=922155
BC00305=922155
BC00306=922151
BC00307=922153
BC00308=922155
BC00309=922155
BC00310=922155
BC00311=922155
BC00312=918747
BC00313=805523
BC00314=697681
BC00315=697681
BC00316=697681
BC00317=733666
BC00318=758324
BC00319=767340
BC00320=794510
BC00321=816578
BC00322=794510
BC00323=758324
BC00324=733666
BC00325=697681
BC00326=697681
BC00327=697681
BC00328=841681
BC00329=841681
BC00330=884227
BC00331=901088
BC00332=895224
BC00333=896289
BC00334=924873
BC00335=936999
BC00336=921975
BC00337=887634
BC00338=824879
BC00339=507816
BC00340=507816
BC00341=552804
BC00342=552804
BC00343=551170
BC00344=493239
BC00345=491979
BC00346=285738
BC00347=285865
BC00348=285441
BC00349=256782
BC00350=258630
BC00351=552804
BC00352=507816
BC00353=507816
BC00354=507816
BC00355=531288
BC00356=531293
BC00357=591240
BC00358=531288
BC00359=507816
BC00360=507816
BC00361=507816
BC00362=507816
BC00363=848972
BC00364=861901
BC00365=963633
BC00366=963633
BC00367=963633
BC00368=963633
BC00369=963633
BC00370=963633
BC00371=963633
BC00372=963633
BC00373=963633
BC00374=963633
BC00375=963633
BC00376=963633
BC00377=963633
BC00378=963633
BC00379=963633
BC00380=902188
BC00381=895372
BC00382=895372
BC00383=895372
BC00384=895372
BC00385=895372
BC00386=840744
BC00387=840744
BC00388=840744
BC00389=840744
BC00390=840744
BC00391=840744
BC00392=779300
BC00393=771332
BC00394=771332
BC00395=771332
BC00396=771332
BC00397=771332
BC00398=717855
BC00399=717855
BC00400=717855
BC00401=717855
BC00402=717855
BC00403=717855
BC00404=656405
BC00405=649173
BC00406=649173
BC00407=649173
BC00408=649173
BC00409=649173
BC00410=594961
BC00411=594961
BC00412=594961
BC00413=594961
BC00414=594961
BC00415=594961
BC00416=594961
BC00417=533517
BC00418=525229
BC00419=525229
BC00420=525229
BC00421=525229
BC00422=525229
BC00423=472073
BC00424=472073
BC00425=472073
BC00426=472073
BC00427=472073
BC00428=472073
BC00429=410629
BC00430=405662
BC00431=402968
BC00432=402968
BC00433=402968
BC00434=402968
BC00435=402968
BC00436=402968
BC00437=349186
BC00438=349186
BC00439=349186
BC00440=349186
BC00441=349186
BC00442=349186
BC00443=336469
BC00444=336469
BC00445=336469
BC00446=336469
BC00447=336469
BC00448=336469
BC00449=336469
BC00450=367602
BC00451=367601
BC00452=367601
BC00453=367601
BC00454=367601
BC00455=367601
BC00456=367601
BC00457=425303
BC00458=425303
BC00459=514953
BC00460=463119
BC00461=419862
BC00462=484962
BC00463=484962
BC00464=395463
BC00465=369502
BC00466=369502
BC00467=369502
BC00468=369502
BC00469=369502
BC00470=369502
BC00471=369502
BC00472=369502
BC00473=368885
BC00474=368885
BC00475=368885
BC00476=368885
BC00477=368885
BC00478=368885
BC00479=419064
BC00480=366918
BC00481=349186
BC00482=353241
BC00483=353241
BC00484=353241
BC00485=353241
BC00486=353241
BC00487=410629
BC00488=409135
BC00489=409135
BC00490=409135
BC00491=409135
BC00492=409135
BC00493=472073
BC00494=476126
BC00495=476126
BC00496=476126
BC00497=476126
BC00498=476126
BC00499=533517
BC00500=532644
BC00501=532644
BC00502=532644
BC00503=532644
BC00504=532644
BC00505=594961
BC00506=599988
BC00507=599988
BC00508=599988
BC00509=599988
BC00510=599988
BC00511=656405
BC00512=653254
BC00513=653254
BC00514=653254
BC00515=653254
BC00516=653254
BC00517=717855
BC00518=721570
BC00519=721570
BC00520=721570
BC00521=721570
BC00522=721570
BC00523=779300
BC00524=777963
BC00525=777963
BC00526=777963
BC00527=777963
BC00528=777963
BC00529=840744
BC00530=843810
BC00531=843810
BC00532=843810
BC00533=843810
BC00534=843810
BC00535=902188
BC00536=900128
BC00537=900128
BC00538=900128
BC00539=900128
BC00540=900128
BC00541=963634
BC00542=965489
BC00543=965489
BC00544=965489
BC00545=965489
BC00546=965489
BC00547=965489
BC00548=965489
BC00549=965489
BC00550=965489
BC00551=965489
BC00552=965489
BC00553=965485
BC00554=965485
BC00555=965485
BC00556=965485
BC00557=931504
BC00558=769966
BC00559=769966
BC00560=716686
BC00561=679663
BC00562=721442
BC00563=721442
BC00564=721439
BC00565=781482
BC00566=781888
BC00567=781888
BC00568=781888
BC00569=781888
BC00570=768943
BC00571=718475
BC00572=718475
BC00573=718475
BC00574=778313
BC00575=778313
BC00576=717855
BC00577=792672
BC00578=792672
BC00579=948195
BC00580=948195
BC00581=957587
BC00582=959389
BC00583=964592
BC00584=964592
BC00585=963973
BC00586=963973
BC00587=963973
BC00588=963828
BC00589=943835
BC00590=792672
BC00591=792672
BC00592=792672
BC00593=887446
BC00594=956264
BC00595=956264
BC00596=969252
BC00597=969265
BC00598=975920
BC00599=977704
BC00600=978415
BC00601=978883
BC00602=978885
BC00603=978885
BC00604=956264
BC00605=887446
BC00606=792672
BC00607=792672
BC00608=700249
BC00609=546214
BC00610=546214
BC00611=546211
BC00612=546211
BC00613=406776
BC00614=406776
BC00615=352261
BC00616=346119
BC00617=406266
BC00618=406266
BC00619=491556
BC00620=546211
BC00621=546214
BC00622=546214
BC00623=507604
BC00624=410782
BC00625=429690
BC00626=375447
BC00627=350474
BC00628=350474
BC00629=408658
BC00630=408658
BC00631=507604
BC00632=546214
BC00633=546214
BC00634=516757
BC00635=591809
BC00636=591809
BC00637=591809
BC00638=591183
BC00639=650353
BC00640=650538
BC00641=650538
BC00642=584003
BC00643=515801
BC00644=520018
BC00645=520018
BC00646=590597
BC00647=593080
BC00648=593080
BC00649=593080
BC00650=652456
BC00651=652559
BC00652=594501
BC00653=537666
BC00654=469748
BC00655=546211
BC00656=830322
BC00657=830322
BC00658=830322
BC00659=890247
BC00660=890396
BC00661=798848
BC00662=798848
BC00663=798848
BC00664=798848
BC00665=832296
BC00666=845010
BC00667=845010
BC00668=904605
BC00669=904704
BC00670=818840
BC00671=818839
BC00672=818839
BC00673=526967
BC00674=334612
BC00675=334612
BC00676=334612
BC00677=350464
BC00678=350464
BC00679=359337
BC00680=359337
BC00681=359337
BC00682=359337
BC00683=359453
BC00684=359337
BC00685=359337
BC00686=359337
BC00687=359337
BC00688=359337
BC00689=358620
BC00690=350464
BC00691=334612
BC00692=334612
BC00693=334612
BC00694=334613
BC00695=501279
BC00696=501279
BC00697=334612
BC00698=334610
BC00699=349510
BC00700=365935
BC00701=365935
BC00702=365934
BC00703=348430
BC00704=348430
BC00705=348430
BC00706=365935
BC00707=349510
BC00708=334610
BC00709=334612
BC00710=334612
BC00711=512789
BC00712=516757
BC00713=526627
BC00714=466969
BC00715=466969
BC00716=466969
BC00717=524647
BC00718=525745
BC00719=525745
BC00720=525745
BC00721=525745
BC00722=473911
BC00723=473911
BC00724=473911
BC00725=532824
BC00726=533743
BC00727=525745
BC00728=525745
BC00729=525747
///POSTYPE BASE
///RECTAN
///RCONF 1,0,0,0,0,0,0,0,0,0,0,0,0,0,0,0,0,0,0,0,0,0,0,0
P00006=0.000,0.000,0.000,0.0000,0.0000,0.0000
///RCONF 0,0,0,0,0,0,0,0,0,0,0,0,0,0,0,0,0,0,0,0,0,0,0,0
P00057=0.000,0.000,2.000,0.0000,0.0000,0.0000
P00058=0.000,0.000,3.000,0.0000,0.0000,0.0000
///RCONF 1,0,0,0,0,0,0,0,0,0,0,0,0,0,0,0,0,0,0,0,0,0,0,0
P00097=0.043,-1.896,1.568,0.0000,0.0000,0.0000
P00098=-0.089,-2.467,4.059,0.0000,0.0000,0.0000
P00099=0.011,-2.380,1.226,0.0000,0.0000,0.0000
P00100=-0.081,2.558,4.482,0.0000,0.0000,0.0000
P00101=0.030,-2.286,2.993,0.0000,0.0000,0.0000
P00102=-0.005,-1.108,1.644,0.0000,0.0000,0.0000
P00103=-0.094,-3.400,4.200,0.0000,0.0000,0.0000
P00104=0.043,-2.127,5.826,0.0000,0.0000,0.0000
P00105=-0.043,0.662,5.286,0.0000,0.0000,0.0000
P00106=-0.018,-2.519,0.237,0.0000,0.0000,0.0000
P00107=-0.008,-4.537,-4.500,0.0000,0.0000,0.0000
P00108=0.014,-3.040,2.637,0.0000,0.0000,0.0000
///RCONF 0,0,0,0,0,0,0,0,0,0,0,0,0,0,0,0,0,0,0,0,0,0,0,0
P00299=-1.404,-0.874,9.133,0.0000,0.0000,0.0000
///RCONF 1,0,0,0,0,0,0,0,0,0,0,0,0,0,0,0,0,0,0,0,0,0,0,0
P00300=-0.036,-1.505,2.318,0.0000,0.0000,0.0000
P00301=0.046,-2.112,7.779,0.0000,0.0000,0.0000
P00302=-0.180,-2.409,6.326,0.0000,0.0000,0.0000
///RCONF 0,0,0,0,0,0,0,0,0,0,0,0,0,0,0,0,0,0,0,0,0,0,0,0
P00303=-0.004,-1.437,-4.584,0.0000,0.0000,0.0000
P00304=0.028,-1.666,-4.234,0.0000,0.0000,0.0000
P00305=-0.003,-1.920,-3.501,0.0000,0.0000,0.0000
P00306=0.015,-2.252,-3.054,0.0000,0.0000,0.0000
P00307=0.019,-2.151,-5.077,0.0000,0.0000,0.0000
P00308=-0.003,-2.092,-4.888,0.0000,0.0000,0.0000
P00309=-0.040,-2.205,-4.992,0.0000,0.0000,0.0000
P00310=-0.006,-2.490,-5.925,0.0000,0.0000,0.0000
P00311=-0.007,-2.079,-5.307,0.0000,0.0000,0.0000
P00312=-0.032,2.202,-7.632,0.0000,0.0000,0.0000
///RCONF 1,0,0,0,0,0,0,0,0,0,0,0,0,0,0,0,0,0,0,0,0,0,0,0
P00349=0.060,0.167,-1.133,0.0000,0.0000,0.0000
///RCONF 0,0,0,0,0,0,0,0,0,0,0,0,0,0,0,0,0,0,0,0,0,0,0,0
P00350=11.519,-0.008,1.149,0.0000,0.0000,0.0000
P00351=13.563,-0.027,-0.653,0.0000,0.0000,0.0000
P00352=13.252,-0.027,-0.827,0.0000,0.0000,0.0000
P00353=10.971,-0.082,0.776,0.0000,0.0000,0.0000
P00354=-0.024,2.508,-1.824,0.0000,0.0000,0.0000
P00355=-0.001,2.528,-1.131,0.0000,0.0000,0.0000
P00356=-0.034,2.921,-0.262,0.0000,0.0000,0.0000
P00357=0.003,3.386,-0.091,0.0000,0.0000,0.0000
P00358=0.014,3.037,-0.020,0.0000,0.0000,0.0000
P00359=-0.005,2.731,0.912,0.0000,0.0000,0.0000
P00360=-0.011,3.412,0.438,0.0000,0.0000,0.0000
P00361=0.018,3.050,1.253,0.0000,0.0000,0.0000
P00362=0.014,2.784,0.148,0.0000,0.0000,0.0000
P00399=-2.449,0.031,8.825,0.0000,0.0000,0.0000
P00400=5.920,-3.503,-0.024,0.0000,0.0000,0.0000
P00401=3.430,-0.021,1.131,0.0000,0.0000,0.0000
P00402=-0.253,1.107,3.062,0.0000,0.0000,0.0000
P00403=-3.666,-0.015,5.328,0.0000,0.0000,0.0000
P00405=2.420,0.007,1.427,0.0000,0.0000,0.0000
P00406=3.513,-0.022,0.429,0.0000,0.0000,0.0000
P00415=-1.781,-1.303,3.250,0.0000,0.0000,0.0000
P00416=0.027,1.119,3.078,0.0000,0.0000,0.0000
//INST
///DATE 2025/03/18 12:24
///ATTR SC,RW
///GROUP1 RB1,BS1
NOP
CALL JOB:MOVE_INTO_TUNNEL
SFTOF
'------------------------
'------------------------
'SPOINA SRODEK DOL
'------------------------
'------------------------
MOVJ C00000 BC00000 VJ=10.00
MOVJ C00001 BC00001 VJ=30.00
'------------------------
'PODLOGA_BEZ_ROZPORKI
'------------------------
'TEST
MOVL C00002 BC00002 V=166.7
MOVL C00003 BC00003 V=166.7 PL=0
REFP 3 C00004 BC00004
CALL JOB:SEARCH-R1
IMOV P0057 V=23.0
SET P0097 P0006
SFTON P0097
REFP 3 C00005 BC00005
CALL JOB:SEARCH-R1
SET P0097 P0006
SFTON P0097
MOVL C00006 BC00006 V=166.7 PL=0
SFTOF
COMM MOVL C00007 BC00007 V=333.3
MOVL C00008 BC00008 V=333.3
MOVL C00009 BC00009 V=166.7 PL=0
REFP 3 C00010 BC00010
CALL JOB:SEARCH-R1
IMOV P0057 V=23.0
SET P0098 P0006
SFTON P0098
REFP 3 C00011 BC00011
CALL JOB:SEARCH-R1
SET P0098 P0006
SFTON P0098
MOVL C00012 BC00012 V=166.7 PL=0
'TEST
SFTOF
MOVJ C00013 BC00013 VJ=20.00
'------------------------
'W38 P
'------------------------
'TEST
MOVL C00014 BC00014 V=166.7
MOVL C00015 BC00015 V=166.7 PL=0
REFP 3 C00016 BC00016
CALL JOB:SEARCH-R1
IMOV P0057 V=23.0
SET P0099 P0006
SFTON P0099
REFP 3 C00017 BC00017
CALL JOB:SEARCH-R1
SET P0099 P0006
SFTON P0099
MOVL C00018 BC00018 V=166.7 PL=0
'TEST
SFTOF
MOVL C00019 BC00019 V=333.3
MOVL C00020 BC00020 V=333.3
'------------------------
'W38 L
'------------------------
'TEST
MOVL C00021 BC00021 V=166.7 PL=0
REFP 3 C00022 BC00022
CALL JOB:SEARCH-R1
IMOV P0057 V=23.0
SET P0100 P0006
SFTON P0100
REFP 3 C00023 BC00023
CALL JOB:SEARCH-R1
SET P0100 P0006
SFTON P0100
MOVL C00024 BC00024 V=166.7 PL=0
'TEST
SFTOF
MOVJ C00025 BC00025 VJ=20.00
'------------------------
'W45 P
'------------------------
MOVL C00026 BC00026 V=166.7 PL=0
REFP 3 C00027 BC00027
CALL JOB:SEARCH-R1
IMOV P0057 V=23.0
SET P0101 P0006
SFTON P0101
REFP 3 C00028 BC00028
CALL JOB:SEARCH-R1
SET P0101 P0006
SFTON P0101
MOVL C00029 BC00029 V=166.7 PL=0
'TEST
SFTOF
MOVJ C00030 BC00030 VJ=20.00
'------------------------
'W45 L
'------------------------
MOVL C00031 BC00031 V=133.3 PL=0
REFP 3 C00032 BC00032
CALL JOB:SEARCH-R1
IMOV P0057 V=23.0
SET P0102 P0006
SFTON P0102
REFP 3 C00033 BC00033
CALL JOB:SEARCH-R1
SET P0102 P0006
SFTON P0102
MOVL C00034 BC00034 V=250.0 PL=0
'TEST
SFTOF
MOVJ C00035 BC00035 VJ=20.00
'------------------------
'W48 P
'------------------------
'TEST
MOVL C00036 BC00036 V=133.3 PL=0
REFP 3 C00037 BC00037
CALL JOB:SEARCH-R1
IMOV P0057 V=23.0
SET P0103 P0006
SFTON P0103
REFP 3 C00038 BC00038
CALL JOB:SEARCH-R1
SET P0103 P0006
SFTON P0103
MOVL C00039 BC00039 V=166.7 PL=0
'TEST
SFTOF
MOVJ C00040 BC00040 VJ=30.00
MOVJ C00041 BC00041 VJ=30.00
MOVJ C00042 BC00042 VJ=30.00
MOVJ C00043 BC00043 VJ=30.00
MOVJ C00044 BC00044 VJ=20.00
MOVL C00045 BC00045 V=250.0
'------------------------
'W48 L
'------------------------
SFTOF
MOVL C00046 BC00046 V=133.3 PL=0
REFP 3 C00047 BC00047
CALL JOB:SEARCH-R1
IMOV P0057 V=23.0
SET P0104 P0006
SFTON P0104
REFP 3 C00048 BC00048
CALL JOB:SEARCH-R1
SET P0104 P0006
SFTON P0104
MOVL C00049 BC00049 V=166.7 PL=0
SFTOF
MOVJ C00050 BC00050 VJ=20.00
'------------------------
'W36 P
'------------------------
MOVL C00051 BC00051 V=133.3 PL=0
REFP 3 C00052 BC00052
CALL JOB:SEARCH-R1
IMOV P0057 V=23.0
SET P0105 P0006
SFTON P0105
REFP 3 C00053 BC00053
CALL JOB:SEARCH-R1
SET P0105 P0006
SFTON P0105
MOVL C00054 BC00054 V=166.7 PL=0
'TEST
SFTOF
MOVJ C00055 BC00055 VJ=20.00
'------------------------
'W36 L
'------------------------
MOVL C00056 BC00056 V=166.7 PL=0
REFP 3 C00057 BC00057
CALL JOB:SEARCH-R1
IMOV P0057 V=23.0
SET P0106 P0006
SFTON P0106
REFP 3 C00058 BC00058
CALL JOB:SEARCH-R1
SET P0106 P0006
SFTON P0106
MOVL C00059 BC00059 V=166.7 PL=0
'TEST
MOVJ C00060 BC00060 VJ=20.00
SFTOF
'------------------------
'W44 P
'------------------------
'TEST
MOVL C00061 BC00061 V=133.3 PL=0
REFP 3 C00062 BC00062
CALL JOB:SEARCH-R1
IMOV P0057 V=23.0
SET P0107 P0006
SFTON P0107
REFP 3 C00063 BC00063
CALL JOB:SEARCH-R1
SET P0107 P0006
SFTON P0107
MOVL C00064 BC00064 V=250.0 PL=0
'TEST
SFTOF
MOVL C00065 BC00065 V=250.0
MOVJ C00066 BC00066 VJ=25.00
MOVJ C00067 BC00067 VJ=25.00
MOVJ C00068 BC00068 VJ=25.00
MOVJ C00069 BC00069 VJ=25.00
MOVJ C00070 BC00070 VJ=30.00
MOVJ C00071 BC00071 VJ=25.00
'------------------------
'W44 L
'------------------------
'TEST
MOVL C00072 BC00072 V=166.7 PL=0
REFP 3 C00073 BC00073
CALL JOB:SEARCH-R1
IMOV P0057 V=23.0
SET P0108 P0006
SFTON P0108
REFP 3 C00074 BC00074
CALL JOB:SEARCH-R1
SET P0108 P0006
SFTON P0108
MOVL C00075 BC00075 V=250.0 PL=0
'TEST
SFTOF
MOVL C00076 BC00076 V=250.0
MOVJ C00077 BC00077 VJ=25.00
IFTHENEXP OT#(1455)=ON ANDEXP OT#(1439)=OFF
	 CALL JOB:TWIN_FRONT_SEARCH_0ST-2_5340
ENDIF
IFTHENEXP OT#(1455)=OFF ANDEXP OT#(1439)=ON
	 CALL JOB:FRONT_SEARCH_0ST-2_5140_TEST
ENDIF
COMM CALL JOB:FRONT_SEARCH_0ST-2_5140
'COMMENT
'COMMENT
'COMMENT
'COMMENT
'COMMENT
'COMMENT
'COMMENT
'COMMENT
COMM MOVJ C00078 BC00078 VJ=20.00
COMM MOVJ C00079 BC00079 VJ=20.00
COMM MOVJ C00080 BC00080 VJ=20.00
COMM 'DODANE
COMM 'SZUKANIE FRONT
COMM '------------------------
COMM '503
COMM '------------------------
COMM MOVL C00081 BC00081 V=333.3
COMM MOVL C00082 BC00082 V=166.7 PL=0
COMM REFP 3 C00083 BC00083
COMM CALL JOB:SEARCH-R1
COMM IMOV P0058 V=16.7
COMM SET P0350 P0006
COMM SFTON P0350
COMM REFP 3 C00084 BC00084
COMM CALL JOB:SEARCH-R1
COMM SET P0350 P0006
COMM SFTON P0350
COMM MOVL C00085 BC00085 V=66.7 PL=0
COMM SFTOF
COMM '------------------------
COMM '------------------------
COMM '502
COMM '------------------------
COMM MOVL C00086 BC00086 V=166.7
COMM MOVL C00087 BC00087 V=66.7 PL=0
COMM REFP 3 C00088 BC00088
COMM CALL JOB:SEARCH-R1
COMM IMOV P0058 V=16.7
COMM SET P0351 P0006
COMM SFTON P0351
COMM REFP 3 C00089 BC00089
COMM CALL JOB:SEARCH-R1
COMM SET P0351 P0006
COMM SFTON P0351
COMM MOVL C00090 BC00090 V=66.7 PL=0
COMM SFTOF
COMM '------------------------
COMM '------------------------
COMM '501
COMM '------------------------
COMM MOVL C00091 BC00091 V=166.7
COMM MOVL C00092 BC00092 V=66.7 PL=0
COMM REFP 3 C00093 BC00093
COMM CALL JOB:SEARCH-R1
COMM IMOV P0058 V=16.7
COMM SET P0352 P0006
COMM SFTON P0352
COMM REFP 3 C00094 BC00094
COMM CALL JOB:SEARCH-R1
COMM SET P0352 P0006
COMM SFTON P0352
COMM MOVL C00095 BC00095 V=66.7 PL=0
COMM SFTOF
COMM '------------------------
COMM '------------------------
COMM '500
COMM '------------------------
COMM MOVL C00096 BC00096 V=166.7
COMM MOVL C00097 BC00097 V=66.7 PL=0
COMM REFP 3 C00098 BC00098
COMM CALL JOB:SEARCH-R1
COMM IMOV P0058 V=16.7
COMM SET P0353 P0006
COMM SFTON P0353
COMM REFP 3 C00099 BC00099
COMM CALL JOB:SEARCH-R1
COMM SET P0353 P0006
COMM SFTON P0353
COMM MOVL C00100 BC00100 V=66.7 PL=0
COMM SFTOF
COMM '------------------------
COMM MOVL C00101 BC00101 V=333.3
COMM MOVL C00102 BC00102 V=333.3
COMM MOVJ C00103 BC00103 VJ=10.00
COMM 'DODANE
COMM MOVJ C00104 BC00104 VJ=10.00
COMM '------------------------
COMM 'SFT402
COMM '------------------------
COMM SFTOF
COMM MOVL C00105 BC00105 V=150.0
COMM MOVL C00106 BC00106 V=66.7 PL=0
COMM REFP 3 C00107 BC00107
COMM CALL JOB:SEARCH-R1
COMM SET P0402 P0006
COMM SFTON P0402
COMM MOVL C00108 BC00108 V=150.0
COMM MOVL C00109 BC00109 V=66.7 PL=0
COMM REFP 3 C00110 BC00110
COMM CALL JOB:SEARCH-R1
COMM SET P0402 P0006
COMM SFTON P0402
COMM MOVL C00111 BC00111 V=133.3
COMM MOVL C00112 BC00112 V=150.0
COMM MOVL C00113 BC00113 V=150.0
COMM MOVL C00114 BC00114 V=66.7 PL=0
COMM REFP 3 C00115 BC00115
COMM CALL JOB:SEARCH-R1
COMM SET P0402 P0006
COMM SFTOF
COMM MOVL C00116 BC00116 V=150.0
COMM '------------------------
COMM 'SFT403
COMM '------------------------
COMM 'START
COMM SFTOF
COMM MOVL C00117 BC00117 V=250.0
COMM MOVL C00118 BC00118 V=133.3 PL=0
COMM REFP 3 C00119 BC00119
COMM CALL JOB:SEARCH-R1
COMM SET P0416 P0006
COMM SFTON P0416
COMM MOVL C00120 BC00120 V=133.3
COMM REFP 3 C00121 BC00121
COMM CALL JOB:SEARCH-R1
COMM SET P0402 P0006
COMM SFTOF
COMM MOVL C00122 BC00122 V=150.0
COMM '------------------------
COMM '------------------------
COMM SFTOF
COMM MOVL C00123 BC00123 V=250.0
COMM MOVL C00124 BC00124 V=133.3 PL=0
COMM REFP 3 C00125 BC00125
COMM CALL JOB:SEARCH-R1
COMM SET P0403 P0006
COMM SFTON P0403
COMM MOVL C00126 BC00126 V=66.7 PL=0
COMM REFP 3 C00127 BC00127
COMM CALL JOB:SEARCH-R1
COMM SET P0403 P0006
COMM SFTOF
COMM MOVL C00128 BC00128 V=150.0
COMM MOVJ C00129 BC00129 VJ=20.00
COMM MOVJ C00130 BC00130 VJ=20.00
COMM '------------------------
COMM 'SFT401
COMM '------------------------
COMM SFTOF
COMM MOVL C00131 BC00131 V=150.0
COMM MOVL C00132 BC00132 V=66.7 PL=0
COMM REFP 3 C00133 BC00133
COMM CALL JOB:SEARCH-R1
COMM SET P0401 P0006
COMM SFTON P0401
COMM MOVL C00134 BC00134 V=66.7 PL=0
COMM REFP 3 C00135 BC00135
COMM CALL JOB:SEARCH-R1
COMM SET P0401 P0006
COMM SFTOF
COMM MOVL C00136 BC00136 V=150.0
COMM 'SFT400
COMM '------------------------
COMM SFTOF
COMM MOVL C00137 BC00137 V=333.3
COMM MOVL C00138 BC00138 V=66.7 PL=0
COMM REFP 3 C00139 BC00139
COMM CALL JOB:SEARCH-R1
COMM SET P0405 P0006
COMM SFTON P0405
COMM MOVL C00140 BC00140 V=66.7 PL=0
COMM REFP 3 C00141 BC00141
COMM CALL JOB:SEARCH-R1
COMM SET P0405 P0006
COMM SFTOF
COMM MOVL C00142 BC00142 V=150.0
COMM 'SFT400
COMM '------------------------
COMM SFTOF
COMM MOVL C00143 BC00143 V=333.3
COMM MOVL C00144 BC00144 V=133.3 PL=0
COMM REFP 3 C00145 BC00145
COMM CALL JOB:SEARCH-R1
COMM SET P0406 P0006
COMM SFTON P0406
COMM MOVL C00146 BC00146 V=66.7 PL=0
COMM REFP 3 C00147 BC00147
COMM CALL JOB:SEARCH-R1
COMM SET P0406 P0006
COMM SFTOF
COMM MOVL C00148 BC00148 V=150.0
COMM 'SFT400
COMM '------------------------
COMM SFTOF
COMM MOVL C00149 BC00149 V=150.0
COMM MOVL C00150 BC00150 V=66.7 PL=0
COMM REFP 3 C00151 BC00151
COMM CALL JOB:SEARCH-R1
COMM SET P0400 P0006
COMM SFTON P0400
COMM MOVL C00152 BC00152 V=150.0
COMM MOVL C00153 BC00153 V=66.7 PL=0
COMM REFP 3 C00154 BC00154
COMM CALL JOB:SEARCH-R1
COMM SET P0400 P0006
COMM SFTON P0400
COMM MOVL C00155 BC00155 V=150.0
COMM MOVL C00156 BC00156 V=150.0
COMM MOVL C00157 BC00157 V=66.7 PL=0
COMM REFP 3 C00158 BC00158
COMM CALL JOB:SEARCH-R1
COMM SET P0400 P0006
COMM SFTOF
COMM MOVL C00159 BC00159 V=83.3
COMM MOVL C00160 BC00160 V=250.0
COMM MOVL C00161 BC00161 V=333.3
COMM MOVL C00162 BC00162 V=66.7 PL=0
COMM REFP 3 C00163 BC00163
COMM CALL JOB:SEARCH-R1
COMM SET P0415 P0006
COMM SFTON P0415
COMM MOVL C00164 BC00164 V=133.3
COMM REFP 3 C00165 BC00165
COMM CALL JOB:SEARCH-R1
COMM SET P0415 P0006
COMM SFTOF
COMM MOVL C00166 BC00166 V=150.0
COMM '------------------------
COMM 'SFT403
COMM '------------------------
COMM 'START
COMM SFTOF
COMM MOVJ C00167 BC00167 VJ=10.00
COMM '------------------------
COMM 'SFT399
COMM '------------------------
COMM 'START
COMM SFTOF
COMM MOVL C00168 BC00168 V=150.0
COMM MOVL C00169 BC00169 V=66.7 PL=0
COMM REFP 3 C00170 BC00170
COMM CALL JOB:SEARCH-R1
COMM SET P0399 P0006
COMM SFTON P0399
COMM MOVL C00171 BC00171 V=66.7 PL=0
COMM REFP 3 C00172 BC00172
COMM CALL JOB:SEARCH-R1
COMM SET P0399 P0006
COMM SFTOF
COMM MOVL C00173 BC00173 V=150.0
COMM MOVJ C00174 BC00174 VJ=20.00
COMM MOVJ C00175 BC00175 VJ=30.00
MOVJ C00176 BC00176 VJ=30.00
MOVJ C00177 BC00177 VJ=30.00
MOVJ C00178 BC00178 VJ=40.00
'WELD
'WELD
MOVJ C00179 BC00179 VJ=20.00
'**********************
'W36
'**********************
MOVL C00180 BC00180 V=500.0
SFTON P0105
MOVL C00181 BC00181 V=166.7 PL=0
SFTOF
MACRO1 MJ#(0) ARGF24
ARCON
SFTON P0106
MOVL C00182 BC00182 V=11.7
ARCOF
SFTOF
MOVJ C00183 BC00183 VJ=15.00
MOVJ C00184 BC00184 VJ=10.00
MOVJ C00185 BC00185 VJ=10.00
MOVJ C00186 BC00186 VJ=10.00
MOVJ C00187 BC00187 VJ=30.00
MOVJ C00188 BC00188 VJ=20.00
MOVJ C00189 BC00189 VJ=10.00
MOVJ C00190 BC00190 VJ=15.00
'**********************
'W38
'**********************
MOVL C00191 BC00191 V=500.0
SFTON P0100
MOVL C00192 BC00192 V=166.7 PL=0
SFTOF
ARCON
SFTON P0099
MOVL C00193 BC00193 V=11.3
ARCOF
SFTOF
'DODANE
MOVL C00194 BC00194 V=500.0
MOVJ C00195 BC00195 VJ=10.00
MOVJ C00196 BC00196 VJ=10.00
MOVJ C00197 BC00197 VJ=10.00
MOVJ C00198 BC00198 VJ=10.00
MOVJ C00199 BC00199 VJ=25.00
COMM '**********************
COMM '**********************
COMM 'POCZATEK SPAWANIA PRZOD
COMM '**********************
COMM '**********************
COMM MOVJ C00200 BC00200 VJ=30.00
COMM MOVL C00201 BC00201 V=416.7
COMM MOVJ C00202 BC00202 VJ=10.00
COMM MOVJ C00203 BC00203 VJ=10.00
COMM MOVL C00204 BC00204 V=150.0
COMM MOVL C00205 BC00205 V=150.0
COMM '**********************
COMM 'W41A SIDE
COMM '**********************
COMM MOVL C00206 BC00206 V=250.0
COMM SFTON P0402
COMM MOVL C00207 BC00207 V=66.7 PL=0
COMM MACRO1 MJ#(0) ARGF14
COMM ARCON
COMM MOVL C00208 BC00208 V=9.2
COMM ARCOF
COMM SFTOF
COMM MOVL C00209 BC00209 V=166.7
COMM '**********************
COMM 'W41A FRONT
COMM '**********************
COMM MOVL C00210 BC00210 V=250.0
COMM SFTON P0350
COMM MOVL C00211 BC00211 V=66.7 PL=0
COMM SFTOF
COMM MACRO1 MJ#(0) ARGF21
COMM ARCON
COMM SFTON P0351
COMM MOVL C00212 BC00212 V=8.3
COMM SFTOF
COMM ARCOF
COMM MOVL C00213 BC00213 V=166.7
COMM '**********************
COMM 'W41B FRONT
COMM '**********************
COMM MOVL C00214 BC00214 V=250.0
COMM SFTON P0352
COMM MOVL C00215 BC00215 V=66.7 PL=0
COMM SFTOF
COMM MACRO1 MJ#(0) ARGF21
COMM ARCON
COMM SFTON P0353
COMM MOVL C00216 BC00216 V=8.3
COMM SFTOF
COMM ARCOF
COMM MOVL C00217 BC00217 V=166.7
COMM MOVL C00218 BC00218 V=100.0
COMM '**********************
COMM 'W41A SIDE
COMM '**********************
COMM SFTON P0400
COMM MOVL C00219 BC00219 V=66.7 PL=0
COMM MACRO1 MJ#(0) ARGF21
COMM ARCON
COMM MOVL C00220 BC00220 V=8.3
COMM ARCOF
COMM SFTOF
COMM MOVL C00221 BC00221 V=166.7
COMM MOVL C00222 BC00222 V=166.7
COMM MOVL C00223 BC00223 V=333.3
COMM MOVJ C00224 BC00224 VJ=20.00
COMM MOVJ C00225 BC00225 VJ=20.00
COMM '**********************
COMM 'W42A.1
COMM '**********************
COMM 'POPRAWIC
COMM MOVL C00226 BC00226 V=500.0
COMM SFTON P0403
COMM MOVL C00227 BC00227 V=66.7 PL=0
COMM MACRO1 MJ#(0) ARGF9
COMM ARCON
COMM MOVL C00228 BC00228 V=9.2
COMM SFTON P0416
COMM MOVL C00229 BC00229 V=9.2
COMM MOVL C00230 BC00230 V=9.2
COMM MOVL C00231 BC00231 V=9.2
COMM SFTON P0402
COMM MOVL C00232 BC00232 V=9.2
COMM MOVL C00233 BC00233 V=9.2
COMM ARCOF
COMM MOVL C00234 BC00234 V=500.0
COMM SFTOF
COMM MOVJ C00235 BC00235 VJ=15.00
COMM 'W42B.1
COMM MOVJ C00236 BC00236 VJ=30.00
COMM MOVJ C00237 BC00237 VJ=30.00
COMM MOVJ C00238 BC00238 VJ=30.00
COMM MOVJ C00239 BC00239 VJ=30.00
COMM '**********************
COMM 'W42B.1
COMM '**********************
COMM MOVL C00240 BC00240 V=500.0
COMM SFTON P0399
COMM MOVL C00241 BC00241 V=66.7 PL=0
COMM MACRO1 MJ#(0) ARGF9
COMM ARCON
COMM SFTON P0415
COMM MOVL C00242 BC00242 V=9.2
COMM MOVL C00243 BC00243 V=9.2
COMM MOVL C00244 BC00244 V=9.2
COMM SFTON P0400
COMM MOVL C00245 BC00245 V=9.2
COMM MOVL C00246 BC00246 V=9.2
COMM ARCOF
COMM MOVL C00247 BC00247 V=500.0
COMM SFTOF
COMM MOVJ C00248 BC00248 VJ=15.00
COMM 'W42A.2
COMM MOVJ C00249 BC00249 VJ=20.00
COMM MOVJ C00250 BC00250 VJ=20.00
COMM MOVJ C00251 BC00251 VJ=20.00
COMM MOVJ C00252 BC00252 VJ=20.00
COMM MOVJ C00253 BC00253 VJ=20.00
COMM '**********************
COMM 'W42A.2
COMM '**********************
COMM MOVL C00254 BC00254 V=500.0
COMM SFTON P0402
COMM MOVL C00255 BC00255 V=66.7 PL=0
COMM SFTOF
COMM MACRO1 MJ#(0) ARGF9
COMM ARCON
COMM SFTON P0402
COMM MOVL C00256 BC00256 V=9.2
COMM ARCOF
COMM MOVL C00257 BC00257 V=166.7
COMM MOVJ C00258 BC00258 VJ=20.00
COMM MOVJ C00259 BC00259 VJ=20.00
COMM MOVL C00260 BC00260 V=166.7
COMM MOVL C00261 BC00261 V=166.7
COMM ARCON
COMM MOVL C00262 BC00262 V=10.8
COMM ARCOF
COMM MOVL C00263 BC00263 V=166.7
COMM MOVJ C00264 BC00264 VJ=10.00
COMM SFTOF
COMM MOVJ C00265 BC00265 VJ=20.00
COMM MOVJ C00266 BC00266 VJ=20.00
COMM MOVJ C00267 BC00267 VJ=20.00
COMM 'W42B.2
COMM MOVJ C00268 BC00268 VJ=20.00
COMM MOVJ C00269 BC00269 VJ=20.00
COMM MOVJ C00270 BC00270 VJ=20.00
COMM MOVJ C00271 BC00271 VJ=20.00
COMM MOVJ C00272 BC00272 VJ=20.00
COMM '**********************
COMM 'W42B.2
COMM '**********************
COMM MOVL C00273 BC00273 V=500.0
COMM SFTON P0400
COMM MOVL C00274 BC00274 V=166.7 PL=0
COMM SFTOF
COMM MACRO1 MJ#(0) ARGF9
COMM ARCON
COMM SFTON P0400
COMM MOVL C00275 BC00275 V=9.2
COMM ARCOF
COMM SFTOF
COMM MOVL C00276 BC00276 V=166.7
COMM MOVL C00277 BC00277 V=166.7
COMM MOVJ C00278 BC00278 VJ=10.00
COMM SFTON P0400
COMM MOVL C00279 BC00279 V=166.7
COMM ARCON
COMM MOVL C00280 BC00280 V=10.8
COMM ARCOF
COMM MOVL C00281 BC00281 V=166.7
COMM MOVL C00282 BC00282 V=500.0
COMM SFTOF
COMM MOVJ C00283 BC00283 VJ=20.00
COMM MOVJ C00284 BC00284 VJ=20.00
COMM 'W42A.3
COMM MOVJ C00285 BC00285 VJ=10.00
COMM MOVJ C00286 BC00286 VJ=20.00
COMM MOVJ C00287 BC00287 VJ=20.00
COMM MOVJ C00288 BC00288 VJ=20.00
COMM '**********************
COMM 'W42A.3
COMM '**********************
COMM MOVL C00289 BC00289 V=500.0
COMM SFTON P0402
COMM MOVL C00290 BC00290 V=166.7 PL=0
COMM MACRO1 MJ#(0) ARGF9
COMM ARCON
COMM MOVL C00291 BC00291 V=9.2
COMM ARCOF
COMM MOVL C00292 BC00292 V=500.0
COMM SFTOF
COMM '**********************
COMM 'W42B.3
COMM '**********************
COMM MOVL C00293 BC00293 V=500.0
COMM SFTON P0400
COMM MOVL C00294 BC00294 V=66.7 PL=0
COMM ARCON
COMM MOVL C00295 BC00295 V=9.2
COMM ARCOF
COMM MOVL C00296 BC00296 V=500.0
COMM SFTOF
COMM MOVJ C00297 BC00297 VJ=10.00
COMM '**********************
COMM 'GORA L
COMM '**********************
COMM MOVL C00298 BC00298 V=500.0
COMM SFTON P0401
COMM MOVL C00299 BC00299 V=66.7 PL=0
COMM MACRO1 MJ#(0) ARGF9
COMM ARCON
COMM MOVL C00300 BC00300 V=11.7
COMM SFTON P0406
COMM MOVL C00301 BC00301 V=11.7
COMM MOVL C00302 BC00302 V=11.7
COMM MOVL C00303 BC00303 V=11.7
COMM ARCOF
COMM MOVL C00304 BC00304 V=500.0
COMM SFTOF
COMM '**********************
COMM 'GORA P
COMM '**********************
COMM MOVL C00305 BC00305 V=166.7
COMM SFTON P0401
COMM MOVL C00306 BC00306 V=166.7 PL=0
COMM ARCON
COMM MOVL C00307 BC00307 V=11.7
COMM SFTON P0405
COMM MOVL C00308 BC00308 V=11.7
COMM MOVL C00309 BC00309 V=11.7
COMM MOVL C00310 BC00310 V=11.7
COMM ARCOF
COMM MOVL C00311 BC00311 V=500.0
COMM SFTOF
COMM MOVJ C00312 BC00312 VJ=10.00
COMM MOVJ C00313 BC00313 VJ=30.00
COMM MOVJ C00314 BC00314 VJ=30.00
COMM 'KONIEC SPAWANIA FRONTU
COMM '**********************
COMM 'W44
COMM '**********************
MOVJ C00315 BC00315 VJ=30.00
MOVJ C00316 BC00316 VJ=30.00
MOVJ C00317 BC00317 VJ=30.00
MOVL C00318 BC00318 V=500.0
SFTON P0107
MOVL C00319 BC00319 V=166.7 PL=0
MACRO1 MJ#(0) ARGF24
ARCON
SFTON P0108
MOVL C00320 BC00320 V=10.8
MOVL C00321 BC00321 V=10.8
ARCOF
SFTOF
MOVL C00322 BC00322 V=500.0
MOVL C00323 BC00323 V=500.0
MOVJ C00324 BC00324 VJ=10.00
MOVJ C00325 BC00325 VJ=10.00
MOVJ C00326 BC00326 VJ=20.00
'**********************
'DODATEK
'**********************
MOVJ C00327 BC00327 VJ=10.00
MOVJ C00328 BC00328 VJ=10.00
MOVJ C00329 BC00329 VJ=20.00
MOVJ C00330 BC00330 VJ=20.00
MOVJ C00331 BC00331 VJ=20.00
MOVL C00332 BC00332 V=333.3
MOVL C00333 BC00333 V=166.7
MACRO1 MJ#(0) ARGF24
SFTON P0108
MOVL C00334 BC00334 V=166.7 PL=0
SFTOF
ARCON
SFTON P0108
MOVL C00335 BC00335 V=10.8
ARCOF
SFTOF
MOVL C00336 BC00336 V=500.0
MOVJ C00337 BC00337 VJ=20.00
MOVJ C00338 BC00338 VJ=30.00
'**********************
'W45
'**********************
MOVJ C00339 BC00339 VJ=30.00
MOVJ C00340 BC00340 VJ=20.00
MOVJ C00341 BC00341 VJ=10.00
MACRO1 MJ#(0) ARGF24
MOVL C00342 BC00342 V=500.0
SFTON P0102
MOVL C00343 BC00343 V=166.7 PL=0
SFTOF
ARCON
SFTON P0101
MOVL C00344 BC00344 V=11.7
ARCOF
SFTOF
MOVL C00345 BC00345 V=500.0
'**********************
'SPOINA_PODLOGA_BRAK_ROZP
'**********************
MOVL C00346 BC00346 V=500.0
MOVL C00347 BC00347 V=500.0
SFTON P0098
MOVL C00348 BC00348 V=166.7 PL=0
SFTOF
ARCON
SFTON P0097
MOVL C00349 BC00349 V=11.3
ARCOF
SFTOF
'DODANE
MOVL C00350 BC00350 V=500.0
MOVJ C00351 BC00351 VJ=10.00
MOVJ C00352 BC00352 VJ=10.00
'**********************
'W48
'**********************
MOVJ C00353 BC00353 VJ=15.00
MOVJ C00354 BC00354 VJ=15.00
MOVJ C00355 BC00355 VJ=15.00
SFTON P0103
MOVL C00356 BC00356 V=166.7 PL=0
SFTOF
ARCON
SFTON P0104
MOVL C00357 BC00357 V=10.8
ARCOF
SFTOF
MOVL C00358 BC00358 V=500.0
MOVJ C00359 BC00359 VJ=15.00
MOVJ C00360 BC00360 VJ=20.00
MOVJ C00361 BC00361 VJ=40.00
'COMMENT
'COMMENT
'COMMENT
IFTHENEXP OT#(1455)=ON ANDEXP OT#(1439)=OFF
	 CALL JOB:TWIN_FRONT_WELD_0ST-2_5340
ENDIF
IFTHENEXP OT#(1455)=OFF ANDEXP OT#(1439)=ON
	 CALL JOB:FRONT_WELD_0ST-2_5140_TEST
ENDIF
'COMMENT
'COMMENT
COMM CALL JOB:FRONT_WELD_0ST-2_5140
MOVJ C00362 BC00362 VJ=40.00
CALL JOB:MOVE_OUT_OF_TUNNEL
CALL JOB:CLEAN-R1
CALL JOB:MOVE_INTO_TUNNEL
MOVJ C00363 BC00363 VJ=30.00 PL=0
'------------------------
'------------------------
'PRAWA STRONA PROFIL GORA
'------------------------
'------------------------
MOVJ C00364 BC00364 VJ=20.00
'------------------------
'W51A L
'------------------------
SFTOF
MOVJ C00365 BC00365 VJ=10.00
MOVL C00366 BC00366 V=66.7 PL=0
REFP 3 C00367 BC00367
CALL JOB:SEARCH-R1
SET P0299 P0006
SFTON P0299
MOVL C00368 BC00368 V=66.7 PL=0
REFP 3 C00369 BC00369
CALL JOB:SEARCH-R1
SET P0299 P0006
SFTON P0299
MOVL C00370 BC00370 V=83.3
MOVL C00371 BC00371 V=166.7 PL=0
REFP 3 C00372 BC00372
CALL JOB:SEARCH-R1
SET P0299 P0006
SFTON P0299
MOVL C00373 BC00373 V=133.3 PL=0
SFTOF
'------------------------
'W51A P
'------------------------
SFTOF
MOVL C00374 BC00374 V=250.0
MOVL C00375 BC00375 V=66.7 PL=0
REFP 3 C00376 BC00376
CALL JOB:SEARCH-R1
SET P0300 P0006
SFTON P0300
MOVL C00377 BC00377 V=66.7 PL=0
REFP 3 C00378 BC00378
CALL JOB:SEARCH-R1
SET P0300 P0006
SFTON P0300
MOVL C00379 BC00379 V=66.7 PL=0
SFTOF
'------------------------
'W54A L
'------------------------
SFTOF
MOVJ C00380 BC00380 VJ=30.00
MOVL C00381 BC00381 V=133.3 PL=0
REFP 3 C00382 BC00382
CALL JOB:SEARCH-R1
SET P0301 P0006
SFTON P0301
MOVL C00383 BC00383 V=66.7 PL=0
REFP 3 C00384 BC00384
CALL JOB:SEARCH-R1
SET P0301 P0006
SFTON P0301
MOVL C00385 BC00385 V=66.7 PL=0
SFTOF
'------------------------
'W54A P
'------------------------
SFTOF
MOVJ C00386 BC00386 VJ=30.00
MOVL C00387 BC00387 V=133.3 PL=0
REFP 3 C00388 BC00388
CALL JOB:SEARCH-R1
SET P0302 P0006
SFTON P0302
MOVL C00389 BC00389 V=66.7 PL=0
REFP 3 C00390 BC00390
CALL JOB:SEARCH-R1
SET P0302 P0006
SFTON P0302
MOVL C00391 BC00391 V=66.7 PL=0
SFTOF
'------------------------
'W50A L
'------------------------
SFTOF
MOVJ C00392 BC00392 VJ=30.00
MOVL C00393 BC00393 V=133.3 PL=0
REFP 3 C00394 BC00394
CALL JOB:SEARCH-R1
SET P0303 P0006
SFTON P0303
MOVL C00395 BC00395 V=66.7 PL=0
REFP 3 C00396 BC00396
CALL JOB:SEARCH-R1
SET P0303 P0006
SFTON P0303
MOVL C00397 BC00397 V=66.7 PL=0
SFTOF
'------------------------
'W50A P
'------------------------
SFTOF
MOVJ C00398 BC00398 VJ=30.00
MOVL C00399 BC00399 V=133.3 PL=0
REFP 3 C00400 BC00400
CALL JOB:SEARCH-R1
SET P0304 P0006
SFTON P0304
MOVL C00401 BC00401 V=66.7 PL=0
REFP 3 C00402 BC00402
CALL JOB:SEARCH-R1
SET P0304 P0006
SFTON P0304
MOVL C00403 BC00403 V=66.7 PL=0
SFTOF
'------------------------
'W53A L
'------------------------
SFTOF
MOVJ C00404 BC00404 VJ=30.00
MOVL C00405 BC00405 V=133.3 PL=0
REFP 3 C00406 BC00406
CALL JOB:SEARCH-R1
SET P0305 P0006
SFTON P0305
MOVL C00407 BC00407 V=66.7 PL=0
REFP 3 C00408 BC00408
CALL JOB:SEARCH-R1
SET P0305 P0006
SFTON P0305
MOVL C00409 BC00409 V=66.7 PL=0
SFTOF
'------------------------
'W53A P
'------------------------
SFTOF
MOVJ C00410 BC00410 VJ=30.00
MOVL C00411 BC00411 V=200.0
MOVL C00412 BC00412 V=66.7 PL=0
REFP 3 C00413 BC00413
CALL JOB:SEARCH-R1
SET P0306 P0006
SFTON P0306
MOVL C00414 BC00414 V=66.7 PL=0
REFP 3 C00415 BC00415
CALL JOB:SEARCH-R1
SET P0306 P0006
SFTON P0306
MOVL C00416 BC00416 V=66.7 PL=0
SFTOF
'------------------------
'W56A L
'------------------------
SFTOF
MOVJ C00417 BC00417 VJ=30.00
MOVL C00418 BC00418 V=133.3 PL=0
REFP 3 C00419 BC00419
CALL JOB:SEARCH-R1
SET P0307 P0006
SFTON P0307
MOVL C00420 BC00420 V=66.7 PL=0
REFP 3 C00421 BC00421
CALL JOB:SEARCH-R1
SET P0307 P0006
SFTON P0307
MOVL C00422 BC00422 V=66.7 PL=0
SFTOF
'------------------------
'W56A P
'------------------------
SFTOF
MOVJ C00423 BC00423 VJ=30.00
MOVL C00424 BC00424 V=133.3 PL=0
REFP 3 C00425 BC00425
CALL JOB:SEARCH-R1
SET P0308 P0006
SFTON P0308
MOVL C00426 BC00426 V=66.7 PL=0
REFP 3 C00427 BC00427
CALL JOB:SEARCH-R1
SET P0308 P0006
SFTON P0308
MOVL C00428 BC00428 V=66.7 PL=0
SFTOF
'------------------------
'W52A L
'------------------------
SFTOF
MOVJ C00429 BC00429 VJ=30.00
MOVL C00430 BC00430 V=250.0
MOVL C00431 BC00431 V=66.7 PL=0
REFP 3 C00432 BC00432
CALL JOB:SEARCH-R1
SET P0309 P0006
SFTON P0309
MOVL C00433 BC00433 V=66.7 PL=0
REFP 3 C00434 BC00434
CALL JOB:SEARCH-R1
SET P0309 P0006
SFTON P0309
MOVL C00435 BC00435 V=66.7 PL=0
SFTOF
'------------------------
'W52A P
'------------------------
SFTOF
MOVJ C00436 BC00436 VJ=5.00
MOVJ C00437 BC00437 VJ=20.00
MOVL C00438 BC00438 V=116.7 PL=0
REFP 3 C00439 BC00439
CALL JOB:SEARCH-R1
SET P0310 P0006
SFTON P0310
MOVL C00440 BC00440 V=66.7 PL=0
REFP 3 C00441 BC00441
CALL JOB:SEARCH-R1
SET P0310 P0006
SFTON P0310
MOVL C00442 BC00442 V=66.7 PL=0
SFTOF
'------------------------
'W55A L
'------------------------
SFTOF
MOVL C00443 BC00443 V=250.0
MOVJ C00444 BC00444 VJ=10.00
MOVL C00445 BC00445 V=66.7 PL=0
REFP 3 C00446 BC00446
CALL JOB:SEARCH-R1
SET P0311 P0006
SFTON P0311
MOVL C00447 BC00447 V=66.7 PL=0
REFP 3 C00448 BC00448
CALL JOB:SEARCH-R1
SET P0311 P0006
SFTON P0311
MOVL C00449 BC00449 V=66.7 PL=0
SFTOF
'------------------------
'W55A P
'------------------------
SFTOF
MOVL C00450 BC00450 V=250.0
MOVL C00451 BC00451 V=166.7
MOVL C00452 BC00452 V=66.7 PL=0
REFP 3 C00453 BC00453
CALL JOB:SEARCH-R1
SET P0312 P0006
SFTON P0312
MOVL C00454 BC00454 V=66.7 PL=0
REFP 3 C00455 BC00455
CALL JOB:SEARCH-R1
SET P0312 P0006
SFTON P0312
MOVL C00456 BC00456 V=66.7 PL=0
MOVL C00457 BC00457 V=166.7
SFTOF
MOVL C00458 BC00458 V=250.0
MOVJ C00459 BC00459 VJ=20.00
MOVJ C00460 BC00460 VJ=20.00
MOVJ C00461 BC00461 VJ=20.00
MOVJ C00462 BC00462 VJ=20.00
MOVJ C00463 BC00463 VJ=20.00
MOVJ C00464 BC00464 VJ=20.00
'------------------------
'------------------------
'LEWA STRONA PROFIL GORA
'------------------------
'------------------------
MOVJ C00465 BC00465 VJ=10.00
'------------------------
'W55B L
'------------------------
SFTOF
MOVJ C00466 BC00466 VJ=10.00
MOVL C00467 BC00467 V=66.7 PL=0
REFP 3 C00468 BC00468
CALL JOB:SEARCH-R1
SET P0349 P0006
SFTON P0349
MOVL C00469 BC00469 V=66.7 PL=0
REFP 3 C00470 BC00470
CALL JOB:SEARCH-R1
SET P0349 P0006
SFTON P0349
MOVL C00471 BC00471 V=66.7 PL=0
SFTOF
MOVJ C00472 BC00472 VJ=10.00
MOVJ C00473 BC00473 VJ=10.00
'------------------------
'W55B P
'------------------------
SFTOF
MOVL C00474 BC00474 V=66.7 PL=0
REFP 3 C00475 BC00475
CALL JOB:SEARCH-R1
SET P0350 P0006
SFTON P0350
MOVL C00476 BC00476 V=66.7 PL=0
REFP 3 C00477 BC00477
CALL JOB:SEARCH-R1
SET P0350 P0006
SFTON P0350
MOVL C00478 BC00478 V=66.7 PL=0
SFTOF
'------------------------
'W52B L
'------------------------
SFTOF
MOVJ C00479 BC00479 VJ=20.00
MOVJ C00480 BC00480 VJ=20.00
MOVL C00481 BC00481 V=150.0
MOVL C00482 BC00482 V=66.7 PL=0
REFP 3 C00483 BC00483
CALL JOB:SEARCH-R1
SET P0351 P0006
SFTON P0351
MOVL C00484 BC00484 V=66.7 PL=0
REFP 3 C00485 BC00485
CALL JOB:SEARCH-R1
SET P0351 P0006
SFTON P0351
MOVL C00486 BC00486 V=66.7 PL=0
SFTOF
'------------------------
'W52B P
'------------------------
SFTOF
MOVJ C00487 BC00487 VJ=30.00
MOVL C00488 BC00488 V=116.7 PL=0
REFP 3 C00489 BC00489
CALL JOB:SEARCH-R1
SET P0352 P0006
SFTON P0352
MOVL C00490 BC00490 V=66.7 PL=0
REFP 3 C00491 BC00491
CALL JOB:SEARCH-R1
SET P0352 P0006
SFTON P0352
MOVL C00492 BC00492 V=66.7 PL=0
SFTOF
'------------------------
'W56B L
'------------------------
SFTOF
MOVJ C00493 BC00493 VJ=30.00
MOVL C00494 BC00494 V=116.7 PL=0
REFP 3 C00495 BC00495
CALL JOB:SEARCH-R1
SET P0353 P0006
SFTON P0353
MOVL C00496 BC00496 V=66.7 PL=0
REFP 3 C00497 BC00497
CALL JOB:SEARCH-R1
SET P0353 P0006
SFTON P0353
MOVL C00498 BC00498 V=66.7 PL=0
SFTOF
'------------------------
'W56B P
'------------------------
SFTOF
MOVJ C00499 BC00499 VJ=30.00
MOVL C00500 BC00500 V=116.7 PL=0
REFP 3 C00501 BC00501
CALL JOB:SEARCH-R1
SET P0354 P0006
SFTON P0354
MOVL C00502 BC00502 V=66.7 PL=0
REFP 3 C00503 BC00503
CALL JOB:SEARCH-R1
SET P0354 P0006
SFTON P0354
MOVL C00504 BC00504 V=66.7 PL=0
SFTOF
'------------------------
'W53B L
'------------------------
SFTOF
MOVJ C00505 BC00505 VJ=30.00
MOVL C00506 BC00506 V=116.7 PL=0
REFP 3 C00507 BC00507
CALL JOB:SEARCH-R1
SET P0355 P0006
SFTON P0355
MOVL C00508 BC00508 V=66.7 PL=0
REFP 3 C00509 BC00509
CALL JOB:SEARCH-R1
SET P0355 P0006
SFTON P0355
MOVL C00510 BC00510 V=66.7 PL=0
SFTOF
'------------------------
'W53B P
'------------------------
SFTOF
MOVJ C00511 BC00511 VJ=30.00
MOVL C00512 BC00512 V=116.7 PL=0
REFP 3 C00513 BC00513
CALL JOB:SEARCH-R1
SET P0356 P0006
SFTON P0356
MOVL C00514 BC00514 V=66.7 PL=0
REFP 3 C00515 BC00515
CALL JOB:SEARCH-R1
SET P0356 P0006
SFTON P0356
MOVL C00516 BC00516 V=66.7 PL=0
SFTOF
'------------------------
'W50B L
'------------------------
SFTOF
MOVJ C00517 BC00517 VJ=30.00
MOVL C00518 BC00518 V=116.7 PL=0
REFP 3 C00519 BC00519
CALL JOB:SEARCH-R1
SET P0357 P0006
SFTON P0357
MOVL C00520 BC00520 V=66.7 PL=0
REFP 3 C00521 BC00521
CALL JOB:SEARCH-R1
SET P0357 P0006
SFTON P0357
MOVL C00522 BC00522 V=66.7 PL=0
SFTOF
'------------------------
'W50B P
'------------------------
SFTOF
MOVJ C00523 BC00523 VJ=30.00
MOVL C00524 BC00524 V=116.7 PL=0
REFP 3 C00525 BC00525
CALL JOB:SEARCH-R1
SET P0358 P0006
SFTON P0358
MOVL C00526 BC00526 V=66.7 PL=0
REFP 3 C00527 BC00527
CALL JOB:SEARCH-R1
SET P0358 P0006
SFTON P0358
MOVL C00528 BC00528 V=66.7 PL=0
SFTOF
'------------------------
'W54B L
'------------------------
SFTOF
MOVJ C00529 BC00529 VJ=30.00
MOVL C00530 BC00530 V=116.7 PL=0
REFP 3 C00531 BC00531
CALL JOB:SEARCH-R1
SET P0359 P0006
SFTON P0359
MOVL C00532 BC00532 V=66.7 PL=0
REFP 3 C00533 BC00533
CALL JOB:SEARCH-R1
SET P0359 P0006
SFTON P0359
MOVL C00534 BC00534 V=66.7 PL=0
SFTOF
'------------------------
'W54B P
'------------------------
SFTOF
MOVJ C00535 BC00535 VJ=30.00
MOVL C00536 BC00536 V=116.7 PL=0
REFP 3 C00537 BC00537
CALL JOB:SEARCH-R1
SET P0360 P0006
SFTON P0360
MOVL C00538 BC00538 V=66.7 PL=0
REFP 3 C00539 BC00539
CALL JOB:SEARCH-R1
SET P0360 P0006
SFTON P0360
MOVL C00540 BC00540 V=66.7 PL=0
SFTOF
'------------------------
'W51B L
'------------------------
SFTOF
MOVJ C00541 BC00541 VJ=30.00
MOVL C00542 BC00542 V=133.3 PL=0
REFP 3 C00543 BC00543
CALL JOB:SEARCH-R1
SET P0361 P0006
SFTON P0361
MOVL C00544 BC00544 V=66.7 PL=0
REFP 3 C00545 BC00545
CALL JOB:SEARCH-R1
SET P0361 P0006
SFTON P0361
MOVL C00546 BC00546 V=66.7 PL=0
SFTOF
'------------------------
'W51B P
'------------------------
SFTOF
MOVL C00547 BC00547 V=150.0
MOVL C00548 BC00548 V=66.7 PL=0
REFP 3 C00549 BC00549
CALL JOB:SEARCH-R1
SET P0362 P0006
SFTON P0362
MOVL C00550 BC00550 V=66.7 PL=0
REFP 3 C00551 BC00551
CALL JOB:SEARCH-R1
SET P0362 P0006
SFTON P0362
MOVL C00552 BC00552 V=83.3
MOVL C00553 BC00553 V=133.3 PL=0
REFP 3 C00554 BC00554
CALL JOB:SEARCH-R1
SET P0362 P0006
SFTON P0362
SFTOF
MOVL C00555 BC00555 V=83.3
MOVL C00556 BC00556 V=250.0
MOVJ C00557 BC00557 VJ=20.00
MOVJ C00558 BC00558 VJ=30.00
MOVJ C00559 BC00559 VJ=10.00
MOVJ C00560 BC00560 VJ=40.00
'**********************
'**********************
'POCZATEK SPAWANIA BOKI
'**********************
'**********************
MOVJ C00561 BC00561 VJ=30.00
MOVJ C00562 BC00562 VJ=20.00
'**********************
'W50A
'**********************
MOVL C00563 BC00563 V=250.0
SFTON P0304
MOVL C00564 BC00564 V=83.3 PL=0
SFTOF
MACRO1 MJ#(0) ARGF10
ARCON
SFTON P0303
MOVL C00565 BC00565 V=10.8
ARCOF
SFTOF
MOVL C00566 BC00566 V=250.0
'W13B
MOVJ C00567 BC00567 VJ=20.00
MOVJ C00568 BC00568 VJ=40.00
MOVJ C00569 BC00569 VJ=20.00
MOVJ C00570 BC00570 VJ=20.00
MOVJ C00571 BC00571 VJ=20.00
'**********************
'W50B
'**********************
MOVL C00572 BC00572 V=250.0
SFTON P0357
MOVL C00573 BC00573 V=166.7 PL=0
SFTOF
MACRO1 MJ#(0) ARGF10
ARCON
SFTON P0358
MOVL C00574 BC00574 V=10.8
ARCOF
SFTOF
MOVL C00575 BC00575 V=250.0
MOVJ C00576 BC00576 VJ=20.00
MOVJ C00577 BC00577 VJ=20.00
MOVJ C00578 BC00578 VJ=20.00
MOVJ C00579 BC00579 VJ=20.00
'**********************
'W51A
'**********************
MOVL C00580 BC00580 V=416.7
MOVL C00581 BC00581 V=416.7
SFTON P0300
MOVL C00582 BC00582 V=166.7 PL=0
SFTOF
MACRO1 MJ#(0) ARGF10
ARCON
SFTON P0299
MOVL C00583 BC00583 V=10.8
MOVL C00584 BC00584 V=10.8
ARCOF
MOVL C00585 BC00585 V=166.7
MOVL C00586 BC00586 V=133.3 PL=0
ARCON
MOVL C00587 BC00587 V=8.3
ARCOF
SFTOF
MOVL C00588 BC00588 V=200.0
MOVL C00589 BC00589 V=333.3
MOVJ C00590 BC00590 VJ=30.00
MOVJ C00591 BC00591 VJ=30.00
MOVJ C00592 BC00592 VJ=30.00
MOVJ C00593 BC00593 VJ=30.00
MOVJ C00594 BC00594 VJ=30.00
'**********************
'W51B
'**********************
MOVL C00595 BC00595 V=416.7
MOVL C00596 BC00596 V=416.7
SFTON P0361
MOVL C00597 BC00597 V=166.7 PL=0
SFTOF
MACRO1 MJ#(0) ARGF10
ARCON
SFTON P0362
MOVL C00598 BC00598 V=10.8
MOVL C00599 BC00599 V=10.8
ARCOF
MOVL C00600 BC00600 V=166.7
MACRO1 MJ#(0) ARGF9
MOVL C00601 BC00601 V=166.7 PL=0
ARCON
MOVL C00602 BC00602 V=8.3
ARCOF
SFTOF
MOVL C00603 BC00603 V=166.7
MOVL C00604 BC00604 V=250.0
MOVJ C00605 BC00605 VJ=30.00
MOVJ C00606 BC00606 VJ=30.00
MOVJ C00607 BC00607 VJ=30.00
MOVJ C00608 BC00608 VJ=40.00
MOVJ C00609 BC00609 VJ=40.00
MOVJ C00610 BC00610 VJ=20.00
MOVJ C00611 BC00611 VJ=20.00
MOVJ C00612 BC00612 VJ=20.00
MOVJ C00613 BC00613 VJ=20.00
MOVJ C00614 BC00614 VJ=20.00
'**********************
'W52A
'**********************
SFTON P0310
MOVL C00615 BC00615 V=250.0
MOVL C00616 BC00616 V=83.3 PL=0
SFTOF
MACRO1 MJ#(0) ARGF10
ARCON
SFTON P0309
MOVL C00617 BC00617 V=10.8
ARCOF
SFTOF
MOVL C00618 BC00618 V=333.3
MOVJ C00619 BC00619 VJ=30.00
MOVJ C00620 BC00620 VJ=30.00
MOVJ C00621 BC00621 VJ=30.00
MOVJ C00622 BC00622 VJ=30.00
MOVJ C00623 BC00623 VJ=30.00
MOVJ C00624 BC00624 VJ=20.00
MOVJ C00625 BC00625 VJ=20.00
MOVJ C00626 BC00626 VJ=20.00
'**********************
'52B
'**********************
MOVL C00627 BC00627 V=250.0
SFTON P0351
MOVL C00628 BC00628 V=83.3 PL=0
SFTOF
MACRO1 MJ#(0) ARGF10
ARCON
SFTON P0352
MOVL C00629 BC00629 V=10.8
ARCOF
MOVL C00630 BC00630 V=333.3
SFTOF
MOVJ C00631 BC00631 VJ=20.00
MOVJ C00632 BC00632 VJ=30.00
MOVJ C00633 BC00633 VJ=30.00
'**********************
'W53A
'**********************
MOVJ C00634 BC00634 VJ=30.00
MOVJ C00635 BC00635 VJ=30.00
MOVJ C00636 BC00636 VJ=10.00
'**********************
'W53A
'**********************
SFTON P0306
MOVL C00637 BC00637 V=250.0
MOVL C00638 BC00638 V=83.3 PL=0
SFTOF
MACRO1 MJ#(0) ARGF10
ARCON
SFTON P0305
MOVL C00639 BC00639 V=10.8
ARCOF
SFTOF
MOVL C00640 BC00640 V=250.0
MOVJ C00641 BC00641 VJ=30.00
MOVJ C00642 BC00642 VJ=30.00
MOVJ C00643 BC00643 VJ=30.00
MOVJ C00644 BC00644 VJ=30.00
MOVJ C00645 BC00645 VJ=30.00
MOVJ C00646 BC00646 VJ=30.00
MOVL C00647 BC00647 V=250.0
'**********************
'W53B
'**********************
SFTON P0355
MOVL C00648 BC00648 V=250.0
MOVL C00649 BC00649 V=83.3 PL=0
SFTOF
MACRO1 MJ#(0) ARGF10
ARCON
SFTON P0356
MOVL C00650 BC00650 V=10.8
ARCOF
SFTOF
MOVL C00651 BC00651 V=333.3
MOVJ C00652 BC00652 VJ=30.00
MOVJ C00653 BC00653 VJ=30.00
MOVJ C00654 BC00654 VJ=30.00
MOVJ C00655 BC00655 VJ=30.00
MOVJ C00656 BC00656 VJ=30.00
'**********************
'W54A
'**********************
SFTON P0302
MOVL C00657 BC00657 V=250.0
MOVL C00658 BC00658 V=83.3 PL=0
SFTOF
MACRO1 MJ#(0) ARGF10
ARCON
SFTON P0301
MOVL C00659 BC00659 V=10.8
ARCOF
SFTOF
MOVL C00660 BC00660 V=333.3
MOVJ C00661 BC00661 VJ=20.00
MOVJ C00662 BC00662 VJ=30.00
MOVJ C00663 BC00663 VJ=30.00
MOVJ C00664 BC00664 VJ=30.00
MOVJ C00665 BC00665 VJ=30.00
'**********************
'W54B
'**********************
SFTON P0359
MOVL C00666 BC00666 V=250.0
MOVL C00667 BC00667 V=83.3 PL=0
SFTOF
MACRO1 MJ#(0) ARGF10
ARCON
SFTON P0360
MOVL C00668 BC00668 V=10.8
ARCOF
MOVL C00669 BC00669 V=333.3
SFTOF
MOVJ C00670 BC00670 VJ=30.00
MOVJ C00671 BC00671 VJ=30.00
MOVJ C00672 BC00672 VJ=30.00
MOVJ C00673 BC00673 VJ=40.00
MOVJ C00674 BC00674 VJ=40.00
MOVJ C00675 BC00675 VJ=10.00
MOVJ C00676 BC00676 VJ=10.00
MOVJ C00677 BC00677 VJ=10.00
MOVJ C00678 BC00678 VJ=15.00
MOVJ C00679 BC00679 VJ=15.00
MOVJ C00680 BC00680 VJ=15.00
MOVJ C00681 BC00681 VJ=15.00
'**********************
'W55A
'**********************
SFTON P0311
MOVL C00682 BC00682 V=166.7 PL=0
SFTOF
MACRO1 MJ#(0) ARGF10
ARCON
SFTON P0312
MOVL C00683 BC00683 V=10.8
MOVL C00684 BC00684 V=10.8
ARCOF
SFTOF
MOVL C00685 BC00685 V=150.0
MOVJ C00686 BC00686 VJ=10.00
MOVJ C00687 BC00687 VJ=10.00
MOVJ C00688 BC00688 VJ=10.00
MOVJ C00689 BC00689 VJ=10.00
MOVJ C00690 BC00690 VJ=10.00
MOVJ C00691 BC00691 VJ=10.00
MOVJ C00692 BC00692 VJ=30.00
MOVJ C00693 BC00693 VJ=30.00
MOVJ C00694 BC00694 VJ=20.00
MOVJ C00695 BC00695 VJ=30.00
MOVJ C00696 BC00696 VJ=20.00
MOVJ C00697 BC00697 VJ=20.00
MOVJ C00698 BC00698 VJ=30.00
MOVJ C00699 BC00699 VJ=20.00
MOVJ C00700 BC00700 VJ=20.00
'**********************
'W55B
'**********************
SFTON P0350
MOVL C00701 BC00701 V=333.3
MOVL C00702 BC00702 V=166.7 PL=0
SFTOF
MACRO1 MJ#(0) ARGF10
ARCON
SFTON P0349
MOVL C00703 BC00703 V=10.8
MOVL C00704 BC00704 V=10.8
ARCOF
SFTOF
MOVL C00705 BC00705 V=66.7
MOVJ C00706 BC00706 VJ=10.00
MOVJ C00707 BC00707 VJ=20.00
MOVJ C00708 BC00708 VJ=20.00
MOVJ C00709 BC00709 VJ=20.00
MOVJ C00710 BC00710 VJ=30.00
MOVJ C00711 BC00711 VJ=50.00
MOVJ C00712 BC00712 VJ=50.00
MOVJ C00713 BC00713 VJ=40.00
MOVJ C00714 BC00714 VJ=20.00
'**********************
'W56A
'**********************
SFTON P0308
MOVL C00715 BC00715 V=333.3
MOVL C00716 BC00716 V=166.7 PL=0
SFTOF
MACRO1 MJ#(0) ARGF10
ARCON
SFTON P0307
MOVL C00717 BC00717 V=10.8
ARCOF
SFTOF
MOVL C00718 BC00718 V=333.3
MOVJ C00719 BC00719 VJ=20.00
MOVJ C00720 BC00720 VJ=30.00
MOVJ C00721 BC00721 VJ=30.00
MOVJ C00722 BC00722 VJ=30.00
'**********************
'W56B
'**********************
SFTON P0353
MOVL C00723 BC00723 V=250.0
MOVL C00724 BC00724 V=166.7 PL=0
SFTOF
MACRO1 MJ#(0) ARGF10
ARCON
SFTON P0354
MOVL C00725 BC00725 V=10.8
ARCOF
SFTOF
MOVL C00726 BC00726 V=333.3
MOVJ C00727 BC00727 VJ=30.00
MOVJ C00728 BC00728 VJ=30.00
MOVJ C00729 BC00729 VJ=30.00
CALL JOB:MOVE_OUT_OF_TUNNEL
CALL JOB:R1-HOME
END
